(* IEC 61131-3 sources: brOscatLib/oscatNetw (part 6) *)

(* ---- SMTP_CLIENT.st ---- *)
FUNCTION_BLOCK SMTP_CLIENT
    (*http://www.oscat.de/images/OSCATNetwork/oscat_netlib121_en.pdf#page=123*)
    CASE step OF

    00:
    	IF ACTIVATE AND NOT activate_last THEN
    		TIMEOUT := MAX(T#10s,TIMEOUT);
    		timeout2 := TIMEOUT + T#1s;
    		timeout3 := TIMEOUT / 2;
    		DONE := FALSE;
    		ip_c_red_disable := FALSE;
    		ERROR_C := DWORD#0;
    		ERROR_T := BYTE#0;
    		FSD.ERROR := BYTE#0;
    		file_delete := FALSE;
    		URL_DATA := STRING_TO_URL(STR:=SERVER,DEFAULT_PROTOCOL:='',DEFAULT_PATH:='/');
    		idx1 := FIND(URL_DATA.USER,'%'); (* % Zeichen auf @ ändern *)
    		IF idx1 > 0 THEN
    			URL_DATA.USER := REPLACE(URL_DATA.USER,'@',1,idx1);
    		END_IF
    		esmtp := LEN(URL_DATA.PASSWORD) > 0; (* SMTP oder ExtendedSMTP *)
    		step := 10;
    	END_IF

    10:
    	IF DNS_CLIENT.DONE THEN
    		step := 20;
    	ELSIF DNS_CLIENT.ERROR <> DWORD#0 THEN
    		ERROR_C := DNS_CLIENT.ERROR;
    		ERROR_T := BYTE#1;
    		step := 980;
    	END_IF

    20:	(* SMTP Kommunikation einrichten *)
    	IF FIND(';SSL;ssl;Ssl', URL_DATA.PROTOCOL) > 1 THEN
    		ssl_mode := BYTE#1;
    		IP_C.C_PORT := SEL(URL_DATA.PORT = WORD#0,URL_DATA.PORT,WORD#465); (* Portnummer eintragen *)
    		IP_C.MAILBOX[16] := BYTE#1; (* SSL Mode freigeben *)
    	ELSIF FIND(';TLS;tls;Tls', URL_DATA.PROTOCOL) > 1 THEN
    		ssl_mode := BYTE#2;
    		IP_C.C_PORT := SEL(URL_DATA.PORT = WORD#0,URL_DATA.PORT,WORD#587); (* Portnummer eintragen *)
    		IP_C.MAILBOX[16] := BYTE#0; (* noch kein SSL Mode*)
    	ELSE
    		ssl_mode := BYTE#0;
    		IP_C.C_PORT := SEL(URL_DATA.PORT = WORD#0,URL_DATA.PORT,WORD#25); (* Portnummer eintragen *)
    		IP_C.MAILBOX[16] := BYTE#0; (* kein SSL Mode*)
    	END_IF

      	IP_C.C_IP := DNS_CLIENT.IP4; (* IP eintragen *)
      	IP_C.C_MODE := BYTE#0; (* Mode: TCP+ACTIV+PORT *)
      	IP_C.TIME_RESET := TRUE; (* Zeitueberwachung rücksetzen *)
      	IP_C.C_ENABLE := TRUE; (* Verbindungsaufbau freigeben *)
      	IP_C.R_OBSERVE := TRUE; (* Empfangsueberwachung *)
    	IP_C.MAILBOX[3] := BYTE#0; (* IP Empfang wieder freigeben *)
    	R_BUF.SIZE := UINT#0;
    	snd_enable := TRUE; (* sofortiges senden erlauben *)
    	snd_idx := 0;
    	step := 30;

    30:
    	IF rcv_state = 220 THEN (* 220 = Service ready *)
    		IF esmtp THEN
    			snd_text := 'EHLO OSCAT'; (* ExtendedSMTP *)

    			str1:= SEL(ssl_mode = BYTE#2,auth_names,auth_names_tls);
    			auth_state := BYTE#0;
    			idx2 := 1900;

    			next_step := 40;
    		ELSE
    			snd_text := 'HELO OSCAT'; (* SMTP *)
    			next_step := 90;
    		END_IF
    		snd_lf_cnt := 1;
    	END_IF

    40:
    	IF rcv_state = 250 THEN
    		(* 250 = Requested mail action okay, complete
    			1. bei manchen Providern wird bei SSL kein AUTH verfahren ausgeben.
    			2. Da die 250 xxx Meldungen vom manchen SMTP-Servern mit mehr als einem Telegramme versendet
    		       werden muss alternativ über Zeitüberwachung eine SSL Sonderbehandlung durchgeführt werden *)
    		IF ssl_mode >= BYTE#1 AND TON_WAIT.ET > T#1s THEN
    			rcv_text := '250-AUTH LOGIN'; (* AUTH vortäuschen *)

            	(*####################  DEBUG-MESSAGE  ###################################*)
    			(*IF _debug_enable THEN
    				LOG_CL.NEW_MSG := 'SMTP: PROBLEM /rcv_text ~1';
    				LOG_CL.PRINTF[1] := rcv_text;
    				LOG_MSG();
    			END_IF*)
    			(*########################################################################*)

    		END_IF

    		IF FIND(rcv_text,'AUTH') > 0 THEN (* BUGFIX  !*)
    			IP_C.MAILBOX[3] := BYTE#1; (* IP Empfang blockieren bis Daten überprüft wurden *)
    			idx1 := 0;
    			step := 50;
    		END_IF

    	END_IF

    50:
    	str2 := ELEMENT_GET(59, idx1, str1); (* Trennzeichen >;< *)

    	(*####################  DEBUG-MESSAGE  ###################################*)
    	(*IF _debug_enable THEN
    		LOG_CL.NEW_MSG := 'ST s1>~1< s2>~2< i1>~2< ~3';
    		LOG_CL.PRINTF[1] := str1;
    		LOG_CL.PRINTF[2] := str2;
    		LOG_CL.PRINTF[3] := INT_TO_STRING(idx1);
    		LOG_CL.PRINTF[4] := rcv_text;
    		LOG_MSG();
    	END_IF*)
    	(*########################################################################*)

    	IF LEN(str2) > 0 THEN
    		IF FIND(rcv_text,str2) > 0 THEN
    			auth_state := BIT_LOAD_B(auth_state, TRUE, idx1);
    			str3 := str2; (* aktuellen AUTH-Type Namen sichern *)
    			idx2 := 1000 + (idx1 * 100); (* Schritt berechnen *)
    		END_IF
    		idx1 := idx1 + 1;
    	ELSE
    		IF auth_state <> BYTE#0 THEN (* AUTH-Type gefunden *)
    			IP_C.MAILBOX[3] := BYTE#0; (* IP Empfang wieder freigeben *)
    			(* mit den jeweiligen Authentifizierung Schritten fortfahren:
    			   1000 = PLAIN / 1100 = LOGIN / 1200 = CRAM-MD5 / 1300 TLS *)
    			step := idx2;
    		ELSE
    			idx1 := 0;
    			rcv_text := '';
    			IP_C.MAILBOX[3] := BYTE#0; (* IP Empfang wieder freigeben *)
    			step := 40; (* warten auf nächste 250 auth meldung *)
    		END_IF
    	END_IF

    	(*####################  DEBUG-MESSAGE  ###################################*)
    	(*IF _debug_enable THEN
    		LOG_CL.NEW_MSG := 'SMTP: /auth ~1 /idx1 ~2 /idx2 ~3 /str3 ~4 /LEN ~5 /step ~6 /str1 ~7';
    		LOG_CL.PRINTF[1] := BYTE_TO_STRING(auth_state);
    		LOG_CL.PRINTF[2] := INT_TO_STRING(idx1);
    		LOG_CL.PRINTF[3] := INT_TO_STRING(idx2);
    		LOG_CL.PRINTF[4] := str3;
    		LOG_CL.PRINTF[5] := INT_TO_STRING(LEN(str2));
    		LOG_CL.PRINTF[6] := INT_TO_STRING(step);
    		LOG_CL.PRINTF[7] := str1;
    		LOG_MSG();
    	END_IF*)
    	(*########################################################################*)

     (* ++++++++++++++++++++++++++++++++++++++++++++++++++++++*)

    90:
    	IF rcv_state = 235 OR rcv_state = 250 THEN (* 235 = Authentication successful / 250 Requested mail action okay *)
    		str2 := MAILFROM;
    		str1 := ELEMENT_GET(59, 0, str2);(* MAILFROM lesen , Trennzeichen >;< *)
    		snd_text := INSERT('MAIL FROM: <>', str1, 12);
    		str3 := REPLACE(snd_text, 'From', 9, 1); (* 'MAIL FROM' durch "From" ersetzen und zwischenspeichern *)
    		next_step := 95;
    		cnt1 := ELEMENT_COUNT(35, MAILTO); (* Trennzeichen >#< , Anzahl der Blöcke bestimmen *)
    		cnt2 := 0;
    	END_IF

    95:
    	IF rcv_state = 250 THEN (* 250 = Requested mail action okay *)
    		IF cnt2 < cnt1 THEN
    			str1 := ELEMENT_GET(35, cnt2, MAILTO);(* Trennzeichen >#< *)
    			cnt3 := ELEMENT_COUNT(59, str1); (* Trennzeichen >;< , Anzahl der Sub-Blöcke bestimmen *)
    			cnt4 := 0;
    			cnt2 := cnt2 + 1;
    			step := 100; (* Blockinhalt auswerten *)
    		ELSE
    			step := 110; (* alle Blöcke bearbeitet *)
    		END_IF
    	END_IF

    100:
    	IF rcv_state = 250 THEN (* 250 = Requested mail action okay *)
    		IF cnt4 < cnt3 THEN
    			str2 := ELEMENT_GET(59, cnt4, str1); (* Trennzeichen >;< *)
    			snd_text := INSERT('RCPT TO: <>', str2, 10);
    			cnt4 := cnt4 + 1;
    			next_step := 100;
    		ELSE
    			step := 95;
    		END_IF
    	END_IF

    110:
    	IF rcv_state = 250 THEN (* 250 = Requested mail action okay *)
    		snd_text := 'DATA';
    		next_step := 120;
    	END_IF

    120:
    	IF rcv_state = 354 THEN (* 354 = Start mail input; end with. *)
    		snd_enable := FALSE;
    		str2 := MAILFROM;
    		str1 := ELEMENT_GET(59, 1, str2);(* Angezeigter Name lesen , Trennzeichen >;< *)
    		IF LEN(str1) > 0 THEN
    			str2 := INSERT('"" ', str1, 1);
    			snd_text := INSERT(str3, str2, 6);
    		ELSE
    			snd_text := str3;
    		END_IF
    		cnt2 := 0;
    		cnt1 := MIN(2,cnt1); (* BlindCopy Block ausblenden *)
    		step := 200;
    	END_IF

    200:
    	IF snd_step = 0 THEN
    		IF cnt2 < cnt1 THEN
    			str1 := ELEMENT_GET(35, cnt2, MAILTO);(* Trennzeichen >#< *)
    			cnt3 := ELEMENT_COUNT(59, str1); (* Trennzeichen >;< , Anzahl der Sub-Blöcke bestimmen *)
    			cnt4 := 0;
    			cnt2 := cnt2 + 1;
    			str3 := SEL(cnt2 = 1,'Cc: <>','To: <>');
    			step := 205; (* Blockinhalt auswerten *)
    		ELSE
    			step := 210; (* alle Blöcke bearbeitet *)
    		END_IF
    	END_IF

    205:
    	IF snd_step = 0 THEN
    		IF cnt4 < cnt3 THEN
    			str2 := ELEMENT_GET(59, cnt4, str1); (* Trennzeichen >;< *)
    			snd_text := INSERT(str3, str2, 5);
    			cnt4 := cnt4 + 1;
    		ELSE
    			step := 200;
    		END_IF
    	END_IF

    210:
    	IF snd_step = 0 THEN
    		snd_text := CONCAT('SUBJECT: ',SUBJECT);
    		step := 220;
    	END_IF

    220:
    	IF snd_step = 0 THEN
    		DTI := UDINT_TO_DT(DT_TO_UDINT(DTI) + INT_TO_UDINT(- DTI_OFFSET * 60)); (* Minuten-Offset auf Sekunden umrechnen und addieren *)
    		IF esmtp THEN (* esmtp Format >Date: Thu, 21 May 1998 05:33:29 -0700< *)
    			str2 := ';Mon;Tue;Wed;Thu;Fri;Sat;Sun';
    			str1 := ELEMENT_GET(59, DAY_OF_WEEK(DT_TO_DATE(DTI)), str2);
    			snd_text := CONCAT('Date: ',str1);
    			str1 := DT_TO_STRF(DTI, 0, ', #H #E #A #N:#R:#T +0000', 1);
    			snd_text := CONCAT(snd_text,str1);
    		ELSE (* SMTP Format >Date: 21 May 98 05:33:29< *)
    			snd_text := DT_TO_STRF(DTI, 0, 'Date: #G #E #B #N:#R:#T', 1);
    		END_IF
    		step := 230;
    	END_IF

    230:
    	IF snd_step = 0 THEN
    		snd_text := 'MIME-Version: 1.0';
    		step := 250;
    	END_IF

    250:
    	IF snd_step = 0 THEN
    		snd_text := 'Content-Type: multipart/mixed;boundary="x"';
    		snd_lf_cnt := 2;
    		step := 260;
    	END_IF

    260:
    	IF snd_step = 0 THEN
    		snd_enable := TRUE;
    		snd_text := 'This is a multi-part message in MIME format.';
    		step := 270;
    	END_IF

    270:
    	IF snd_step = 0 THEN
    		snd_enable := FALSE;
    		snd_text := '--x';
    		snd_lf_cnt := 1;
    		step := 280;
    	END_IF

    280:
    	IF snd_step = 0 THEN
    		snd_text := 'Content-Type: text/plain; format=flowed; charset="iso-8859-1";';
    		snd_text := CONCAT(snd_text,' reply-type=original'); (* PCWORX kann nur konstanten mit max 80 zeichen *)
    		step := 290;
    	END_IF

    290:
    	IF snd_step = 0 THEN
    		snd_text := 'Content-Transfer-Encoding: 8bit';
    		snd_lf_cnt := 2;
    		step := 300;
    	END_IF

    300:
    	IF snd_step = 0 THEN
    		snd_enable := TRUE;
    		snd_text := BODY;
    		snd_lf_cnt := 2;
    		step := 310;
    	END_IF

    310:
    	IF snd_step = 0 THEN
    		cnt1 := ELEMENT_COUNT(59, FILES) - 1; (* Anzahl der Dateien *)
    		step := 400;
    	END_IF

    (* +++++++++++++ File-Attachment ++++++++++++ *)
    400:
    	IF cnt1 >= 0 THEN
    		str1 := ELEMENT_GET(59, cnt1, FILES);
    		FILE_PATH_SPLIT(FILENAME:=str1,X:=fpd); (* Datei-Path zerlegen *)
    		IF fpd.FILENAME = '#DEL#' THEN
    			file_delete := TRUE;
    		ELSE
    			step := 410;
    		END_IF
    		cnt1 := cnt1 - 1;
    	ELSE
    		step := 800;
    	END_IF

    410:
    	IF snd_step = 0 THEN
    		snd_enable := FALSE;
    		snd_text := '--x';
    		snd_lf_cnt := 1;
    		step := 420;
    	END_IF

    420:
    	IF snd_step = 0 THEN
    		snd_text := 'Content-Transfer-Encoding: BASE64';
    		str2 := CONCAT(fpd.FILENAME,'"');
    		step := 430;
    	END_IF

    430:
    	IF snd_step = 0 THEN
    		snd_text := CONCAT('Content-Type: application/octet-stream; name="',str2);
    		step := 440;
    	END_IF

    440:
    	IF snd_step = 0 THEN
    		snd_enable := TRUE;
    		snd_text := CONCAT('Content-Disposition: attachment; filename="',str2);
    		snd_lf_cnt := 2;
    		step := 450;
    	END_IF

    450:
    	IF snd_step = 0 THEN
    		FSD.FILENAME := str1; (* Dateiname *)
    		FSD.OFFSET := UDINT#0; (* Start bei Dateianfang *)
    		step := 460;
    	END_IF

    460:
    	FSD.MODE := BYTE#1; (* vorhandene Datei zum lesen öffnen *)
    	F_BUF.SIZE := b64_max; (* maximale länge einlesen *)
    	idx1 := 0;
    	idx2 := 0;
    	step := 470;

    470:
    	IF FSD.MODE = BYTE#0 AND FSD.ERROR = BYTE#0 THEN
    		last_block := FSD.FILE_SIZE = FSD.OFFSET;
    		b64_size1 := MIN(48,UINT_TO_INT(F_BUF.SIZE) - idx1);
    		IF b64_size1 > 0 THEN
    			idx3 := b64_size1 - 1;
    			FOR i1 := 0 TO idx3 DO (* daten in BASE64 buffer kopieren *)
    				b64_buf1[i1] := F_BUF.BUFFER[idx1];
    				idx1 := idx1 + 1;
    			END_FOR
    			BASE64_ENCODE_STREAM( SIZE1:= b64_size1, BUF1:= b64_buf1, BUF2:= b64_buf2, SIZE2=> b64_size2); (* BASE64 Kodierung *)
    			idx3 := b64_size2 - 1;
    			FOR i1 := 0 TO idx3 DO (* Daten aus BASE64 buffer kopieren *)
    				S_BUF.BUFFER[idx2] := b64_buf2[i1];
    				idx2 := idx2 + 1;
    			END_FOR
    			b64_lf := TRUE;
    			(*####################  DEBUG-MESSAGE  ###################################*)
    			(*IF _debug_enable THEN
    				LOG_CL.NEW_MSG := 'B64: FILE ~1 /SIZE ~2 /OFF ~3 /BSIZE ~4 /idx1 ~5 /idx2 ~6';
    				LOG_CL.PRINTF[1] := FSD.FILENAME;
    				LOG_CL.PRINTF[2] := UDINT_TO_STRING(FSD.FILE_SIZE);
    				LOG_CL.PRINTF[3] := UDINT_TO_STRING(FSD.OFFSET);
    				LOG_CL.PRINTF[4] := INT_TO_STRING(b64_size1);
    				LOG_CL.PRINTF[5] := INT_TO_STRING(idx1);
    				LOG_CL.PRINTF[6] := INT_TO_STRING(idx2);
    				LOG_MSG();
    			END_IF*)
    			(*########################################################################*)
    		ELSE
    			b64_lf := last_block;
    			step := 480; (* block beendet  *)
    		END_IF
    		IF b64_lf THEN
    			S_BUF.BUFFER[idx2] := BYTE#16#0D;
    			idx2 := idx2 + 1;
    			S_BUF.BUFFER[idx2] := BYTE#16#0A;
    			idx2 := idx2 + 1;
    		END_IF
    		(*####################  DEBUG-MESSAGE  ###################################*)
    		(*IF _debug_enable THEN
    			LOG_CL.NEW_MSG := 'B64: exit ~1 /SIZE ~2 /OFF ~3 /eof ~4 /lf_cnt ~5';
    			LOG_CL.PRINTF[1] := FSD.FILENAME;
    			LOG_CL.PRINTF[2] := UDINT_TO_STRING(FSD.FILE_SIZE);
    			LOG_CL.PRINTF[3] := UDINT_TO_STRING(FSD.OFFSET);
    			LOG_CL.PRINTF[4] := BOOL_TO_STRING(last_block);
    			LOG_CL.PRINTF[5] := INT_TO_STRING(snd_lf_cnt);
    			LOG_MSG();
    		END_IF*)
    		(*########################################################################*)
    	END_IF

    480:
    	S_BUF.SIZE := INT_TO_UINT(idx2); (* Daten senden *)
    	(*####################  DEBUG-MESSAGE  ###################################*)
    	(*IF _debug_enable THEN
    		LOG_CL.NEW_MSG := 'B64: tcp_send ~1';
    		LOG_CL.PRINTF[1] := INT_TO_STRING(idx2);
    		LOG_MSG();
    	END_IF*)
    	(*########################################################################*)
    	step := 490;

    490:
    	IF S_BUF.SIZE = UINT#0 THEN (* warten bis alle daten gesendet sind *)
    		step := SEL(last_block ,460,400);
    	END_IF

    (* ++++++++++++++++++++++++++++++++++++++++ *)

    800:
    	IF snd_step = 0 THEN
    		snd_enable := FALSE;
    		snd_text := '--x--';
    		snd_lf_cnt := 2;
    		step := 810;
    	END_IF

    810:
    	IF snd_step = 0 THEN
    		snd_enable := TRUE;
    		snd_text := '.';
    		snd_lf_cnt := 1;
    		step := 820;
    	END_IF

    820:
    	IF rcv_state = 250 THEN (* 250 = Requested mail action okay *)
    		snd_text := 'QUIT';
    		ip_c_red_disable := TRUE;
    		next_step := 830;
    	END_IF

    830:
    	IF rcv_state = 221  OR TON_WAIT.ET > timeout3 THEN (* 221 = Service closing transmission channel *)
    		step := 900;
    	END_IF

    (* ================================================== *)

    900:
    	IF file_delete THEN (* Dateien nach transfer löschen *)
    		cnt1 := ELEMENT_COUNT(59, FILES) - 1; (* Trennzeichen >;< , Anzahl der Dateien *)
    		step := 910;
    	ELSE
    		step := 950;
    	END_IF

    910:
    	IF FSD.MODE = BYTE#0 AND FSD.ERROR = BYTE#0 THEN
    		IF cnt1 >= 0 THEN
    			str1 := ELEMENT_GET(59, cnt1, FILES); (* Trennzeichen >;< *)
    			IF str1 <> '#DEL#' THEN
    				FSD.FILENAME := str1;
    				FSD.MODE := BYTE#4; (* File Remove *)
    			END_IF
    			cnt1 := cnt1 - 1;
    		ELSE
    			step := 950;
    		END_IF
    	END_IF

    950:
    	DONE := TRUE;
    	step := 980;

    980:
    	IP_C.C_ENABLE := FALSE; (* SMTP Steuerkanal schliessen *)
    	S_BUF.SIZE := UINT#0;
    	R_BUF.SIZE := UINT#0;
    	IP_C.MAILBOX[3] := BYTE#0; (* IP Empfang wieder freigeben *)
    	snd_step := 0;
    	next_step := 0;
    	FSD.MODE := BYTE#5; (* Datei schliessen *)
    	step := 990;

    990:
    	IF IP_C.C_STATE = BYTE#0 AND FSD.FILE_OPEN = FALSE THEN
    		step := 0;
    	END_IF

    (*  +++++++++++++++++ Authentifizierung +++++++++++++++++ *)

    (* PLAIN ++++++++++++++++++++++++++++++++++++++++++++++++++++++++++ *)

    1000:
    	snd_text := CONCAT('AUTH',str3);
    	snd_lf_cnt := 1;
     	step := 1010;

    1010:
    	IF rcv_state = 334 THEN (* 334 = Authentifizierung  *)
    		cnt1 := LEN(URL_DATA.USER);
    		cnt2 := LEN(URL_DATA.PASSWORD);
    		IF cnt1 + cnt2 <= 46 THEN (* USER + PASSWORD dürfen zusammen maximal 46 Zeichen haben *)
    			b64_buf1[0] := BYTE#0;
    			FOR i1 := 1 TO cnt1 DO
    				b64_buf1[i1] := CODE(URL_DATA.USER, i1);
    			END_FOR
    			b64_size1 := cnt1 + 1;
    			b64_buf1[b64_size1] := BYTE#0;
    			b64_size1 := b64_size1 + 1;
    			FOR i1 := 1 TO cnt2 DO
    				b64_buf1[b64_size1] := CODE(URL_DATA.PASSWORD, i1);
    				b64_size1 := b64_size1 + 1;
    			END_FOR
    			BASE64_ENCODE_STREAM( SIZE1:= b64_size1, BUF1:= b64_buf1, BUF2:= b64_buf2, SIZE2=> b64_size2); (* BASE64 Kodierung *)
    			idx1 := b64_size2 - 1;
    			FOR i1 := 0 TO idx1 DO
    				S_BUF.BUFFER[i1] := b64_buf2[i1];
    			END_FOR
    			S_BUF.BUFFER[b64_size2] := BYTE#16#0D;
    			b64_size2 := b64_size2 + 1;
    			S_BUF.BUFFER[b64_size2] := BYTE#16#0A;
    			b64_size2 := b64_size2 + 1;
    			S_BUF.SIZE := INT_TO_UINT(b64_size2);
    			rcv_state := 0;
    		END_IF
    		step := 90;
    	END_IF

    (* LOGIN ++++++++++++++++++++++++++++++++++++++++++++++++++++++++++ *)

    1100:
    	snd_text := CONCAT('AUTH',str3);
    	snd_lf_cnt := 1;
     	step := 1110;

    1110:
    	IF rcv_state = 334 THEN (* 334 = Authentifizierung  *)
    		b64_str1 := URL_DATA.USER;
    		b64_start := TRUE; (* BASE64 kodierung von Username *)
    		step := 1120;
    	END_IF

    1120:
    	IF b64_start AND b64_done THEN
    		b64_start := FALSE;
    		snd_text := b64_str2;
    		next_step := 1130;
    	END_IF

    1130:
    	IF rcv_state = 334 THEN (* 334 = Password:  *)
    		b64_str1 := URL_DATA.PASSWORD;
    		b64_start := TRUE; (* BASE64 kodierung von Password *)
    		step := 1140;
    	END_IF

    1140:
    	IF b64_start AND b64_done THEN
    		b64_start := FALSE;
    		snd_text := b64_str2;
    		next_step := 90;
    	END_IF

    (* CRAM-MD5  ++++++++++++++++++++++++++++++++++++++++++++++++++++++++++
    (Challenge-Response Authentication Mechanism, Message Digest 5) Authentifizierung auf Basis von MD5-HMAC-Algorithmus. *)

    1200:
    	snd_text := CONCAT('AUTH',str3);
    	snd_lf_cnt := 1;
     	step := 1210;

    1210:
    	IF rcv_state = 334 THEN (* 334 = Authentifizierung  *)
    		md5_b64_ts := RIGHT(rcv_text,LEN(rcv_text) - 4);
    		md5_user := URL_DATA.USER;
    		md5_password := URL_DATA.PASSWORD;
    		MD5_RUN := TRUE;
    		step := 1220;
    	END_IF

    1220:
    	MD5_CRAM_AUTH(RUN:=MD5_RUN,USERNAME:=md5_user,PASSWORD:=md5_password,B64_TS:=md5_b64_ts,AUTH_KEY:=md5_auth_key);
    	IF NOT MD5_RUN THEN
    		snd_text := md5_auth_key;
    		step := 90;
    	END_IF

    (* STARTTLS  ++++++++++++++++++++++++++++++++++++++++++++++++++++++++++ *)

    1300:
    	snd_text := 'STARTTLS';
    	snd_lf_cnt := 1;
     	step := 1310;

    1310:
    	IF rcv_state = 220 THEN (* 220 = Service ready - Ready to start TLS *)
    		IP_C.MAILBOX[16] := BYTE#1; (* SSL/TLS aktivieren *)
    		step := 1320;
    	END_IF

    1320:
    	IF IP_C.MAILBOX[16] = BYTE#2 THEN (* warten bis SSL/TLS aktiviert wurde *)
    		step := 30; (* ganzer Ablauf von vorne beginnen *)
    	END_IF

    (* keine Authentifizierung gefunden +++++++++++++++++++++++++++++++ *)
    1900: ; (* Auf Laufzeitfehler warten *)

    END_CASE
    (* ++++++++++++++++++++++++++++++++++++++++++++++++++++++++++ *)
    IF step >= 30 THEN
    	IF R_BUF.SIZE > UINT#0 THEN (* Daten wurden empfangen ? *)
    		idx1 := UINT_TO_INT(R_BUF.SIZE);
    		REPEAT (* zeilenterminierung erkennen und echtes TEXT-Ende bestimmen *)
    			idx1 := idx1 - 1;
    		UNTIL idx1 = 0 OR R_BUF.BUFFER[idx1] >= BYTE#32 (* TRUE = EXIT *)
    		END_REPEAT
    		FOR i1 := 0 TO idx1 DO (* bei multiline alle CRLF durch >< ersetzen *)
    			IF R_BUF.BUFFER[i1] < BYTE#32 THEN
    				R_BUF.BUFFER[i1] := BYTE#94; (* >< *)
    			END_IF
    		END_FOR
    		rcv_text := BUFFER_TO_STRING(PT:=ADR(R_BUF.BUFFER),SIZE:=idx1+1,START:=0,STOP:=STRING_LENGTH-1);
    		IF LEN(rcv_text) >= 3 THEN (* Statuscode prüfen und auswerten *)
    			rcv_s := LEFT(rcv_text,3);
    			IF IS_NUM(STR:=rcv_s) THEN (* enthält nur Zahlen ? *)
    				rcv_state := STRING_TO_INT(rcv_s);
    			END_IF
    			IP_C.R_OBSERVE := FALSE;
    		END_IF
    		R_BUF.SIZE := UINT#0; (* daten löschen *)

    		(*####################  DEBUG-MESSAGE  ###################################*)
    		(*IF _debug_enable THEN
    			LOG_CL.NEW_MSG := 'RCV: >~1<';
    			LOG_CL.PRINTF[1] := rcv_text;
    			LOG_MSG();
    		END_IF*)
    		(*########################################################################*)

    	END_IF
    END_IF

    (* automatisches Datensenden *)

    CASE snd_step OF

    00:
    	IF LEN(snd_text) > 0 THEN

    		(*####################  DEBUG-MESSAGE  ###################################*)
    		(*IF _debug_enable THEN
    			LOG_CL.NEW_MSG := 'SND: >~1< /lf ~2';
    			LOG_CL.PRINTF[1] := snd_text;
    			LOG_CL.PRINTF[2] := INT_TO_STRING(snd_lf_cnt);
    			LOG_MSG();
    		END_IF*)
    		(*########################################################################*)

    		_STRING_TO_BUFFER(str:=snd_text,pos:=snd_idx,pt:=ADR(S_BUF.BUFFER),size:=SIZEOF(S_BUF.BUFFER)); (* String in puffer kopieren *)
    		snd_idx := snd_idx + LEN(snd_text);
    		FOR i1 := 1 TO snd_lf_cnt DO
    			S_BUF.BUFFER[snd_idx] := BYTE#16#0D;
    			snd_idx := snd_idx + 1;
    			S_BUF.BUFFER[snd_idx] := BYTE#16#0A;
    			snd_idx := snd_idx + 1;
    		END_FOR
    		snd_text := '';
    		rcv_state := 9999; (* letzen SMTP Status löschen *)

    		IF snd_enable THEN
    			S_BUF.SIZE := INT_TO_UINT(snd_idx); (* Sendelänge eintragen *)
    			R_BUF.SIZE := UINT#0; (* Empfangsbuffer rücksetzen *)
    			IP_C.R_OBSERVE := step <= 120 OR step >= 820;
    			snd_idx := 0;
    			snd_step := 10;
    		END_IF
    	END_IF

    10:
    	IF S_BUF.SIZE = UINT#0 THEN (* warten bis alle daten gesendet sind *)
    		IF next_step <> 0 THEN
    			step := next_step;
    			next_step := 0;
    		END_IF
    		snd_step := 0;
    	END_IF

    END_CASE

    (* Globale Fehlerbehandlung für Haupt-Routine *)
    IF ERROR_T = BYTE#0 AND step > 20 THEN (* noch kein Fehler gespeichert und Hauptroutine aktiv *)

    	IF IP_C.ERROR > DWORD#0 AND IP_C.C_ENABLE AND NOT IP_C.TIME_RESET THEN  (* IP Control 1 *)
    		IF ip_c_red_disable = FALSE OR IP_C.ERROR <> DWORD#16#FD000000 THEN
    			ERROR_C := IP_C.ERROR;
    			ERROR_T := BYTE#2;
    			step := 980;
    		END_IF
    	END_IF

    	IF FSD.MODE = BYTE#0 THEN
    		IF FSD.ERROR > BYTE#0 THEN
    			ERROR_C := BYTE_TO_DWORD(FSD.ERROR);
    			ERROR_T := BYTE#4; (* Dateizugriff *)
    			step := 980;
    		END_IF
    	END_IF
    END_IF

    IF TON_WAIT.Q THEN (* Ablaufstörung - Schrittkette *)
    	ERROR_C := SHL(INT_TO_DWORD(step),16) OR INT_TO_DWORD(rcv_state); (* aktuellen Schritt und letzten SMTP Status eintragen *)
    	ERROR_T := BYTE#5;
    	step := 980;
    END_IF

    (* ######################################################## *)

    DNS_CLIENT(IP_C:=IP_C, S_BUF:=S_BUF, R_BUF:=R_BUF, DOMAIN:=URL_DATA.DOMAIN, IP4_DNS:= DNS_IP4, ACTIVATE:=step=10); (* DNS-Client *)
    IPC(IP:= DWORD#0, PORT:= WORD#0 , TIME_OUT:= TIMEOUT, IP_C:= IP_C, S_BUF:= S_BUF, R_BUF:= R_BUF); (* SMTP Steuerkanal *)
    FS(FSD:=FSD,PT:=F_BUF); (* FILE_SERVER *)
    BASE64_ENCODE_STR(RUN:= b64_start, str1:= b64_str1, str2:= b64_str2, DONE=> b64_done); (* BASE64 kodierung *)

    TON_WAIT(IN:=step = last_step AND step > 0,PT:=timeout2);
    last_step := step;
    activate_last := ACTIVATE;
    BUSY := step <> 0;

    (* revision history
    ks	01. jan. 2011	rev 1.0
    	original version
    ks	06. apr. 2011	rev 1.1
    	list_len und list_get durch element_count und element_get ersetzt
    ks	11. may 2011	rev 1.2
    	ip_control - remote disconnect error ausblenden, und sonderbehandlung für pcworx
    ks	30. may 2011	rev 1.3
    	fehler bei receive-TIMEOUT
    ks	05. may. 2012	rev 1.4
    	FileServer AutoClose entfernt und Fehler im Alias Name korrigiert
    ks	06. apr. 2013	rev 1.5
    	Fehler bei Authorisierungsabfrage bei 1&1 Provider behoben
    ks	22. feb. 2016	rev 1.6
    	integration SSL/TLS
    ks	11. aug. 2016	rev 1.7
    	bugfix: Find SSL/TLS String in URL_DATA.PROTOCOL
    *)
END_FUNCTION_BLOCK

(* ---- SNTP_CLIENT.st ---- *)
FUNCTION_BLOCK SNTP_CLIENT
    (*http://www.oscat.de/images/OSCATNetwork/oscat_netlib121_en.pdf#page=127*)
    (* Domain Name System (query) *)
    tx := T_PLC_MS(); (* read system time *)

    CASE state OF
    00: (* auf positive Flanke SET warten *)
    	DONE_P := FALSE;
    	IF ACTIVATE AND NOT activate_last THEN
    		ip4_stored := IP4; (* aktuelle IP4 speichern *)
    		state := 10;
    		ERROR := DWORD#0;
    		ip_state := BYTE#1; (* Anmelden *)
    		(*####################  DEBUG-MESSAGE  ###################################*)
    		(*IF _debug_enable THEN
    			LOG_CL.NEW_MSG := 'SNTP: S00 START';
    			LOG_MSG();
    		END_IF*)
    		(*########################################################################*)
    	END_IF

    10: (* Bei IP_Control anmelden und auf freigabe warten *)
    	IF ip_state = BYTE#3 THEN

    		S_BUF.BUFFER[00] := BYTE#16#1B;
    		FOR i := 1 TO 47 DO
    			S_BUF.BUFFER[i] := BYTE#16#00;
    		END_FOR

    		last := tx; (* aktuellen time wert sichern *)
    		state := 30;

    		(* IP Datenverkehr einrichten *)
    		IP_C.C_PORT := WORD#123; (* Portnummer eintragen *)
    		IP_C.C_IP := ip4_stored; (* IP eintragen *)
    		IP_C.C_MODE := BYTE#1; (* Mode: UDP+AKTIV+PORT+IP *)
    		IP_C.C_ENABLE := TRUE; (* Verbindungsaufbau freigeben *)
    		IP_C.TIME_RESET := TRUE; (* Zeitueberwachung rücksetzen *)
    		IP_C.R_OBSERVE := TRUE; (* Datenempfang ueberwachen *)
    		S_BUF.SIZE := UINT#48; (* Sendelänge eintragen *)
    		R_BUF.SIZE := UINT#0; (* Empfangslänge rücksetzen *)
        		(*####################  DEBUG-MESSAGE  ###################################*)
        		(*IF _debug_enable THEN
          			LOG_CL.NEW_MSG := 'SNTP: S10 SEND';
          			LOG_MSG();
        		END_IF*)
        		(*########################################################################*)
    	END_IF

    30:
    	IF IP_C.ERROR <> DWORD#00 THEN
    		ERROR := IP_C.ERROR;
    		S_BUF.SIZE := UINT#0;
    		R_BUF.SIZE := UINT#0;
    		state := 0;
        		(*####################  DEBUG-MESSAGE  ###################################*)
        		(*IF _debug_enable THEN
          			LOG_CL.NEW_MSG := 'SNTP: S30 ERROR ~1';
          			LOG_CL.PRINTF[1] := DWORD_TO_STRING(ERROR);
          			LOG_MSG();
        		END_IF*)
        		(*########################################################################*)

    	ELSIF S_BUF.SIZE = UINT#0 AND R_BUF.SIZE >= UINT#48 THEN (* länge der empfangenen Daten prüfen *)

    		(* Umrechnung SNTP Timestamp Base 1900-01-01 -> Unix 1970-01-01 = +2208988800 sekunden*)
    		UDT := DWORD_TO_DT(DWORD_OF_BYTE(R_BUF.BUFFER[40],R_BUF.BUFFER[41],R_BUF.BUFFER[42],R_BUF.BUFFER[43]) - DWORD#2208988800);

    		(* Original-Sekundenanteile sind als 32 Bit Fractal dargestellt *)
    		(* ms nur mit veringerte Auflösung berechnen 1/65535 -> Highword verwenden *)
    		XMS := DWORD_TO_INT(SHR(DINT_TO_DWORD(WORD_TO_DINT(WORD_OF_BYTE(R_BUF.BUFFER[44],R_BUF.BUFFER[45])) * DINT#1000),16));
    		(* Zeitdifferenz (Laufzeitfehler) zwischen Send und Receive /2 teilen und addieren *)
    		XMS := XMS + DWORD_TO_INT(SHR(tx - last,1));

    		UDT := DWORD_TO_DT(DT_TO_DWORD(UDT) + (XMS / 1000)); (* sekundenanteile der Zeitdifferenz zu UDT aufrechnen *)
    		XMS := XMS MOD 1000;  (* ms übernehmen *)
    		state := 0;
    		DONE_P := TRUE;
        		(*####################  DEBUG-MESSAGE  ###################################*)
        		(*IF _debug_enable THEN
            			LOG_CL.NEW_MSG := 'SNTP: S30 OK';
            			LOG_MSG();
        		END_IF*)
        		(*########################################################################*)

    	END_IF

    	IF state = 0 THEN
    		IP_C.R_OBSERVE := FALSE; (* Datenempfang ueberwachen *)
    		ip_state := BYTE#4;
    	END_IF

    END_CASE

    activate_last := ACTIVATE; (* letzten Status sichern zur Flankenerkennung *)

    (* IP_FIFO *)
    IP_FIFO(FIFO:=IP_C.FIFO,state:=ip_state,ID:=ip_id);

    (* revision history
    ks	18. oct. 2008	rev 1.0
    	original version

    ks	20. oct. 2009	rev 1.1
    	Networkbuffer und Buffer-funktionen auf Basis 0

    *)

    (***************************************************************************************)
    (*               SNTP Datenstruktur
                                      1                   2                   3
                  0 1 2 3 4 5 6 7 8 9 0 1 2 3 4 5 6 7 8 9 0 1 2 3 4 5 6 7 8 9 0 1
                 +-+-+-+-+-+-+-+-+-+-+-+-+-+-+-+-+-+-+-+-+-+-+-+-+-+-+-+-+-+-+-+-+
    Byte: 01-04  |LI | VN  |Mode |    Stratum    |     Poll      |   Precision   |
                 +-+-+-+-+-+-+-+-+-+-+-+-+-+-+-+-+-+-+-+-+-+-+-+-+-+-+-+-+-+-+-+-+
    Byte: 05-08  |                          Root  Delay (32 Bit)                 |
                 +-+-+-+-+-+-+-+-+-+-+-+-+-+-+-+-+-+-+-+-+-+-+-+-+-+-+-+-+-+-+-+-+
    Byte: 09-12  |                       Root  Dispersion (32 Bit)               |
                 +-+-+-+-+-+-+-+-+-+-+-+-+-+-+-+-+-+-+-+-+-+-+-+-+-+-+-+-+-+-+-+-+
    Byte: 13-16  |                     Reference Identifier (32 Bit)             |
                 +-+-+-+-+-+-+-+-+-+-+-+-+-+-+-+-+-+-+-+-+-+-+-+-+-+-+-+-+-+-+-+-+
    Byte: 17-24  |                    Reference Timestamp (64 Bit)               |
                 +-+-+-+-+-+-+-+-+-+-+-+-+-+-+-+-+-+-+-+-+-+-+-+-+-+-+-+-+-+-+-+-+
    Byte: 25-32  |                    Originate Timestamp (64 Bit)               |
                 +-+-+-+-+-+-+-+-+-+-+-+-+-+-+-+-+-+-+-+-+-+-+-+-+-+-+-+-+-+-+-+-+
    Byte: 33-40  |                     Receive Timestamp (64 Bit)                |
                 +-+-+-+-+-+-+-+-+-+-+-+-+-+-+-+-+-+-+-+-+-+-+-+-+-+-+-+-+-+-+-+-+
    Byte: 41-48  |                     Transmit Timestamp (64 Bit)               |
                 +-+-+-+-+-+-+-+-+-+-+-+-+-+-+-+-+-+-+-+-+-+-+-+-+-+-+-+-+-+-+-+-+
    Byte: 49-52  |                 Key Identifier (optional) (32 Bit)            |
                 +-+-+-+-+-+-+-+-+-+-+-+-+-+-+-+-+-+-+-+-+-+-+-+-+-+-+-+-+-+-+-+-+
    Byte: 53-68  |                 Message Digest (optional) (128 Bit)           |
                 +-+-+-+-+-+-+-+-+-+-+-+-+-+-+-+-+-+-+-+-+-+-+-+-+-+-+-+-+-+-+-+-+

    *)

    (*
    Worldwide NTP-Server

    NIST-Zeitserver
    • time-a.nist.gov
    129.6.15.28
    NIST, Gaithersburg, Maryland
    • time-a.nist.gov
    129.6.15.28
    NIST, Gaithersburg, Maryland
    • time-a.timefreq.bldrdoc.gov
    132.163.4.101 (Stand: 1. Dezember 1999)
    NIST, Boulder, Colorado
    • time-b.timefreq.bldrdoc.gov
    132.163.4.102 (Stand: 1. Dezember 1999)
    NIST, Boulder, Colorado
    • time-c.timefreq.bldrdoc.gov
    132.163.4.103 (Stand: 1. Dezember 1999)
    NIST, Boulder, Colorado
    • utcnist.colorado.edu
    128.138.140.44
    University of Colorado, Boulder
    • time.nist.gov
    192.43.244.18
    NCAR, Boulder, Colorado
    • time-nw.nist.gov
    131.107.1.10
    Microsoft, Redmond, Washington
    • nist1.dc.certifiedtime.com
    216.200.93.8
    Abovnet, North Virginia
    • nist1.datum.com
    209.0.72.7
    Datum, San Jose, Kalifornien
    • nist1.nyc.certifiedtime.com
    208.184.49.129
    Abovnet, New York City
    • nist1.sjc.certifiedtime.com
    207.126.103.202
    Abovnet, San Jose, Kalifornien

    Zeitserver der ersten Ebene
    Sortiert nach Standort:
    Nordamerika
    • Palo Alto, Kalifornien: Systems Research Center, Compaq Computer Corp.
    204.123.2.72: usno.pa-x.dec.com; CNAME: navobs1.pa-x.dec.com
    Servicebereich: US-Zeitzonen PST (Pacific Standard Time) und MST (Mountain Standard Time)
    • Marina del Rey, Kalifornien: USC Information Sciences Institute
    128.9.176.30: timekeeper.isi.edu
    Servicebereich: CalRen2- und Los Nettos-Bereich
    • Washington, DC: U.S. Naval Observatory
    192.5.41.41: tock.usno.navy.mil
    192.5.41.40: tick.usno.navy.mil
    Servicebereich: NSFNET
    • Ottawa, Ontario, Kanada: National Research Council of Canada
    time.chu.nrc.ca
    Servicebereich: Kanada
    • Raleigh, North Carolina: North Carolina state University
    152.1.58.124: terrapin.csc.ncsu.edu
    Servicebereich: Südosten der USA
    • Cambridge, Massachusetts: MIT Information Systems
    18.72.0.3: bitsy.mit.edu
    Servicebereich: NSFNET- und NEARnet-Bereich
    • Cambridge, Massachusetts: MIT
    18.26.4.105: bonehed.lcs.mit.edu
    Servicebereich: Osten der USA
    • Palo Alto, Kalifornien: Internet Software Consortium
    192.5.5.250: clock.isc.org
    Servicebereich: BARRnet, Alternet-West und CIX-West
    • Cambridge, Massachusetts: Open Software Foundation
    130.105.4.59: clock.osf.org
    Servicebereich: NSFNET- und NEARnet-Bereich
    • Palo Alto, Kalifornien: ViaNet Communications
    209.81.9.7: clock.via.net
    • Cleveland, Ohio: Lewis Research Center (NASA)
    128.156.1.43: lerc-dns.lerc.nasa.gov
    Servicebereich: NSFNET und OARNET
    • Colorado Springs, Colorado: Schriever AFB
    204.34.198.40: navobs1.usnogps.navy.mil; CNAME: tick.usnogps.navy.mil
    204.34.198.41: navobs1.usnogps.navy.mil; CNAME: tock.usnogps.navy.mil
    Servicebereich: US-Zeitzonen PST (Pacific Standard Time) und MST (Mountain Standard Time)
    • St. Louis, Missouri: Washington University
    128.252.19.1: navobs1.usnogps.navy.mil; CNAME: tick.wustl.edu
    Servicebereich: US-Zeitzone CST (Central Standard Time)
    • Research Triangle Park, North Carolina: MCNC
    192.101.21.1: ncnoc.ncren.net
    Servicebereich: NC-REN-Bereich (North Carolina Research and Education Network)
    • Cupertino, Kalifornien: HP
    192.6.38.127: ntp-cup.external.hp.com
    Servicebereich: USA Westküste
    • Newark, Delaware: Conectiv Communications
    138.39.7.20: ntp1.delmarva.com
    Servicebereich: Cable & Wireless Network (früher MCInet)
    • University Park, Pennsylvania: Penn state University
    128.118.46.3: otc1.psu.edu
    Servicebereich: NSFNET, PREPNET und JvNCnet

    Europa
    • Borowiec, Polen: Astrogeodynamical Observatory, Space Research Centre
    150.254.183.15: vega.cbk.poznan.pl
    Servicebereich: Polen und Europa
    • Stockholm, Schweden: Stupi AB
    192.36.143.151: Time2.Stupi.SE
    Servicebereich: Europa
    • Turin, Italien: IEN Galileo Ferraris
    193.204.114.1: time.ien.it
    Servicebereich: Italien und Europa
    • Zürich, Schweiz: Integrated Systems Laboratory , Eidgenössischen Technischen Hochschule Zürich
    129.132.2.21: swisstime.ethz.ch
    Servicebereich: Schweiz und Europa
    • Turin, Italien: CSTV of National Research Council
    150.145.33.1: tempo.cstv.to.cnr.it
    Servicebereich: Italien und Europa
    • Erlangen, Deutschland: Universität Erlangen-Nürnberg
    ntp0.fau.de; ntp1.fau.de; ntp2.fau.de;
    ntps1-0.uni-erlangen.de; ntps1-1.uni-erlangen.de; ntps1-2.uni-erlangen.de
    Servicebereich: Deutschland und Europa
    • Berlin, Deutschland: Technische Universität Berlin
    130.149.17.21: ntps1-0.cs.tu-berlin.de
    130.149.17.8: ntps1-1.cs.tu-berlin.de
    Servicebereich: Deutschland und Europa
    • Deutschland
    131.173.17.7: ntps1-1.rz.Uni-Osnabrueck.DE
    Servicebereich: Deutschland und Europa
    • Schweden
    192.36.143.150: Time1.Stupi.SE
    Servicebereich: SUnet und NORDUnet Schweden

    Fernost und pazifische Randgebiete
    • Hong Kong: Chinesische Universität von Hong Kong.
    137.189.6.18: clock.cuhk.edu.hk
    Servicebereich: Hong Kong (China) und Südostasien
    • Fukuoka, Japan: Universität Fukuoka
    133.100.9.2: clock.nc.fukuoka-u.ac.jp
    133.100.11.8: clock.tl.fukuoka-u.ac.jp
    Servicebereich: Japan und pazifischer Raum

    Australien
    • Melbourne, Australien: University of Melbourne
    128.250.36.2: ntp.cs.mu.OZ.AU
    Servicebereich: Australien und Neuseeland

    Zeitserver der zweiten Ebene
    Nach geographischem Standort sortiert:
    Nordamerika
    NTP-Zeitserver: • Quebec, Kanada: Canadian Meteorological Center
    ntp1.cmc.ec.gc.ca; ntp2.cmc.ec.gc.ca
    Servicebereich: Ostkanada
    • Ontario, Kanada: National Research Council of Canada
    time.chu.nrc.ca; time.nrc.ca
    Servicebereich: Kanada
    • Saskatchewan, Kanada: University of Regina
    142.3.100.15: timelord.uregina.ca
    Servicebereich: Kanada
    • Ontario, Kanada: University of Toronto
    tick.utoronto.ca; tock.utoronto.ca
    Servicebereich: Ostkanada
    • Mexiko: Audiotel-Büro
    ntp2a.audiotel.com.mx; ntp2c.audiotel.com.mx; ntp2b.audiotel.com.mx
    Servicebereich: Avantel, MCINet und Mexiko
    • Santa Cruz, Kalifornien: Scruz-net, inc.
    165.227.1.1: ns.scruz.net
    Servicebereich: Westen der USA
    • San Diego, Kalifornien: UCSD Academic Computing Services/Network Operations
    132.239.254.49: ntp.ucsd.edu
    Servicebereich: CERFNET; NSFNET, SDSC-Bereich, und nahegelegene Bereiche
    • Quincy, Kalifornien
    ntp1.mainecoon.com; ntp2.mainecoon.com
    Servicebereich: Nordamerika
    • Newark, Delaware: University of Delaware
    128.175.1.3: louie.udel.edu
    Servicebereich: CAIRN, Abilene und vBNS
    • Atlanta, Georgia: CNSG
    ntp.shorty.com
    Servicebereich: Südwesten der USA
    • Kennesaw, Georgia: PeachNet
    rolex.peachnet.edu; timex.peachnet.edu
    Servicebereich: PeachNet (Georgia) und Südwesten der USA
    • Urbana-Champaign, Illinois: University of Illinois
    ntp-0.cso.uiuc.edu; ntp-1.cso.uiuc.edu; ntp-2.cso.uiuc.edu
    Servicebereich: CICNET, Mittlerer Westen und NCSA-Bereich
    • Chicago, Illinois: Argonne National Laboratory
    ntp-1.mcs.anl.gov; ntp-2.mcs.anl.gov
    Servicebereich: NSF/ANSNet, CICNet, NetIllinois und ESNet
    • West Lafayette, Indiana: Purdue University
    gilbreth.ecn.purdue.edu; harbor.ecn.purdue.edu; molecule.ecn.purdue.edu
    Servicebereich: NSFNET- und CICNET-Bereich
    • Manhattan, Kansas: KansasNet OnLine Services
    199.240.130.1: ntp1.kansas.net
    199.240.130.12: ntp2.kansas.net
    Servicebereich: Zentral-USA und Great Plains
    • Boston, Massachusetts: UMass-Boston CS dept.
    158.121.104.4: timeserver.cs.umb.edu
    Servicebereich: Neuengland
    • Minneapolis/St Paul, Minnesota: University of Minnesota
    ns.nts.umn.edu; nss.nts.umn.edu
    Servicebereich: CICNET-Bereich
    • Columbia, Missouri: University of Missouri-Columbia
    128.206.206.12: everest.cclabs.missouri.edu
    Servicebereich: MOREnet
    • Omaha, Nebraska: Radiks Internet Access
    205.138.126.83: allison.radiks.net
    Servicebereich: Mittlerer Westen, USA
    • Las Vegas, Nevada: University of Nevada System Computing Services
    131.216.1.101: cuckoo.nevada.edu
    Servicebereich: NevadaNet, NSFNET und SDSC-Bereich
    • Las Vegas, Nevada: UNLV College of Engineering
    tick.cs.unlv.edu; tock.cs.unlv.edu
    Servicebereich: Sprintnet
    • New York City, New York: Columbia University
    ntp.ctr.columbia.edu
    Servicebereich: Sprintlink und NYSERnet
    • Ithaca, New York: Cornell University
    192.35.82.50: ntp0.cornell.edu
    Servicebereich: NSFNET und NYSER-Bereich
    • New York, New York: Morningside Campus, Columbia University
    sundial.columbia.edu
    Servicebereich: NYSERnet
    • New York City, New York: Columbia University Computer Science Department
    timex.cs.columbia.edu
    Servicebereich: PSINET; NSFNET, und NYSER-Bereich
    • Norman, Oklahoma: University of Oklahoma
    129.15.22.8: constellation.ecn.uoknor.edu
    Servicebereich: Midnet
    • Coos Bay, Oregon: Koala Computers
    207.48.109.6: tick.koalas.com
    Servicebereich: Nordwesten der USA
    • University Park, Pennsylvania: Penn state University
    128.118.25.3: clock.psu.edu
    Servicebereich: Internet2, vBNS, CERFnet(AT&T IP Services), PSC/NCNE und CASC
    • Pittsburgh, Pennsylvania: Pittsburgh Supercomputing Center
    128.182.58.100: fuzz.psc.edu
    Servicebereich: NSFNET und PSC-Bereich
    • Pittsburgh, Pennsylvania: Carnegie Mellon Electrical and Computer Engineering
    ntp-1.ece.cmu.edu; ntp-2.ece.cmu.edu
    Servicebereich: PREPNET und PSC-Bereich
    • Dallas, Texas: Cox School of Business, Southern Methodist University
    129.119.80.126: ntp.cox.smu.edu
    Servicebereich: NSFNET und SESQUI-Bereich
    • Hughes Springs, Texas: First National Bank
    209.144.20.76: ntp.fnbhs.com
    Servicebereich: Nordosten Texas
    • Houston, Texas: Baylor College of Medicine
    128.249.1.10: ntp.tmc.edu
    Servicebereich: NSFNET und SESQUI-Bereich
    • College Station, Texas: Texas A&M University
    165.91.52.110: ntp5.tamu.edu
    Servicebereich: NSFNET, SESQUI-Bereich, THEnet und TAMUSDSN
    • Plano, Texas: Greyware Automation Products
    tick.greyware.com; tock.greyware.com
    Servicebereich: Südzentral-USA
    • Blacksburg, Virginia: Virginia Tech Computing Center
    ntp-1.vt.edu; ntp-2.vt.edu
    Servicebereich: Südwesten der USA
    • Arlington, Virginia: Center for Seismic Studies
    140.162.1.3: ntp.cmr.gov
    Servicebereich: NSFNET und SURA-Bereich
    • Richland, Washington: Washington state University
    192.31.216.30: clock.tricity.wsu.edu
    Servicebereich: NSFNET und NorthWestNet
    • Washington, USA: Mill Creek
    time.ultimeth.net
    Servicebereich: Nordwesten der USA
    • Wisconsin, USA: Computer Science Department, University of Wisconsin-Madison
    ntp1.cs.wisc.edu; ntp2.cs.wisc.edu; ntp3.cs.wisc.edu
    Servicebereich: USA und jeder andere

    Südamerika
    • Buenos Aires, Argentinien: Network Access Point
    200.49.40.1: CNAME: tick.nap.com.ar
    200.49.32.1: CNAME: tock.nap.com.ar
    Servicebereich: Argentinien
    • Buenos Aires, Argentinien: Sinectis S.A.
    time.sinectis.com.ar
    Servicebereich: Argentinien
    • Brasilien: Brazilian Research Network
    200.144.121.33: ntp.cais.rnp.br
    Servicebereich: Brasilien
    • Venezuela: VELUG, Grupo de Usuarios Linux de Venezuela
    150.185.192.250: ntp.linux.org.ve
    Servicebereich: Arica

    Europa
    • Zürich, Schweiz: Eidgenössischen Technischen Hochschule Zürich
    129.132.98.11: bernina.ethz.ch
    Servicebereich: Schweiz und Europa
    • Standort: Kopenhagen, Dänemark, Europa
    clock.netcetera.dk; clock2.netcetera.dk
    Servicebereich: Dänemark, Skandinavien und Nordeuropa
    • Spanien: Altea
    slug.ctv.es
    Servicebereich: Spanien
    • Pieksamaki, Finnland: Keski-Savon Oppimiskeskus
    tick.keso.fi; tock.keso.fi
    Servicebereich: Finnland
    • Meudon, Frankreich: Observatoire de Paris-Meudon
    ntp.obspm.fr
    Servicebereich: Frankreich und Europa
    • Lyon, Frankreich: CISM
    ntp.univ-lyon1.fr
    Servicebereich: Frankreich, Schweiz, Italien und Europa
    • Paris, Frankreich: VIA, Ecole Centrale
    138.195.130.70: ntp.via.ecp.fr
    Servicebereich: Frankreich und Europa
    • Budapest, Ungarn: KFKI Research Institute for Particle and Nuclear Physics
    148.6.0.1: time.kfki.hu
    Servicebereich: HUNGARNET
    • Italien: Net4u Srl, Vercelli, Italien
    195.32.52.129: ntps.net4u.it
    Servicebereich: Italien
    • Oslo, Norwegen: Universität Oslo
    129.240.64.3: fartein.ifi.uio.no
    Servicebereich: NORDUnet
    • Oslo, Norwegen: Alcanet International
    time.alcanet.no
    Servicebereich: Europa
    • Krakau, Polen: Academic Computer Centre
    149.156.4.11: info.cyf-kr.edu.pl
    Servicebereich: Polen und Europa
    • Lund, Schweden: Lund Institute of Technology
    130.235.20.3: ntp.lth.se
    Servicebereich: Schweden und NORDUnet
    • Ljubljana, Slowenien: Institute of Biophysics, University of Ljubljana
    biofiz.mf.uni-lj.si 193.2.69.11
    Servicebereich: Slowenien und Europa
    • Ljubljana, Slowenien: Hydrometeorological Institute of Slovenia
    hmljhp.rzs-hm.si
    Servicebereich: Slowenien und Europa
    • Ljubljana, Slowenien: Academic and Research Network of Slovenia
    ntp1.arnes.si; ntp2.arnes.si
    Servicebereich: Slowenien und Europa
    • Ljubljana, Slowenien: J. Stefan Institute
    time.ijs.si
    Servicebereich: Slowenien und Europa

    Britische Inseln
    • Dublin, Irland: School of Mathematics, Trinity College
    ntp.cs.tcd.ie; ntp.maths.tcd.ie; ntp.tcd.ie
    Servicebereich: Irland und Großbritannien
    • Glasgow, Schottland: Strathclyde University
    ntp.cs.strath.ac.uk
    Servicebereich: Großbritannien, Europa und andere
    • Cambridge, Großbritannien
    ntp0.uk.uu.net; ntp1.uk.uu.net;
    ntp2.uk.uu.net
    Servicebereich: UUNET (in Großbritannien früher auch als PIPEX bekannt) und Großbritannien.
    • Manchester, England: University of Manchester
    ntp2a.mcc.ac.uk; ntp2b.mcc.ac.uk;
    ntp2c.mcc.ac.uk; ntp2d.mcc.ac.uk
    Servicebereich: Großbritannien
    • Buckinghamshire, Großbritannien: Wibble U.K., Aylesbury
    tick.tanac.net
    Servicebereich: Großbritannien

    Asien
    • Moskau, Russland: Landau Institute for Theoretical Physics
    193.233.9.7: ntp.landau.ac.ru
    Servicebereich: Russland
    • Russland: Pushchino (bei Moskau)
    194.149.67.130: ntp.psn.ru
    Servicebereich: Russland
    • Chernogolovka, Russland: Chernogolovka Scientific Center (bei Moskau)
    193.233.46.10: sign.chg.ru
    Servicebereich: Russland

    Fernost und pazifische Randgebiete
    • Tokyo, Japan: Cyber Fleet, Inc.
    203.139.30.195: ntp.cyber-fleet.net
    Servicebereich: Japan und Ostasien
    • Seoul, Korea: Inet, Inc.
    time.nuri.net
    Servicebereich: Korea, Japan, Hong Kong und Ostasien
    • Hamilton, Neuseeland: Universität Waikato
    truechimer.waikato.ac.nz; truechimer1.waikato.ac.nz;
    truechimer2.waikato.ac.nz; truechimer3.waikato.ac.nz
    Servicebereich: Neuseeland
    • Singapur und Philippinen:
    ntp.shim.org
    Servicebereich: Singapur

    Afrika
    • Lagos, Nigeria: Supernet300
    ntp.supernet300.com
    Servicebereich: Westafrika (hauptsächlich nigerischer NITEL-Backbone)
    • Pietermaritzburg, Südafrika: Natal University
    143.128.82.200: ntp.cs.unp.ac.za
    Servicebereich: Südafrika

    Australien
    • Adelaide, Südaustralien: University of Adelaide
    129.127.28.4: augean.eleceng.adelaide.edu.au
    129.127.40.3: ntp.adelaide.edu.au
    203.21.37.18: ntp.saard.net
    Servicebereich: AARNet
    • Carlton, Victoria, Australien: eSec Limited
    203.21.84.4: time.esec.com.au

    *)
END_FUNCTION_BLOCK

(* ---- SNTP_SERVER.st ---- *)
FUNCTION_BLOCK SNTP_SERVER
    (*http://www.oscat.de/images/OSCATNetwork/oscat_netlib121_en.pdf#page=128*)
    (* Domain Name System (query) *)
    tx := T_PLC_MS(); (* read system time *)

    CASE state OF

    00: (* Warten auf Freigabe *)
    	IF ENABLE THEN
    		state := 10;
    		ip_state := BYTE#1; (* Anmelden *)
        		(*####################  DEBUG-MESSAGE  ###################################*)
        		(*IF _debug_enable THEN
          			LOG_CL.NEW_MSG := 'SNTP_SERVER: S00 START';
          			LOG_MSG();
        		END_IF*)
        		(*########################################################################*)
    	END_IF

    10: (* Bei IP_Control anmelden und auf freigabe warten *)
    	IF ip_state = BYTE#3 THEN
    		(* IP Datenverkehr einrichten *)
    		IP_C.C_PORT := WORD#123; (* Portnummer eintragen *)
    		IP_C.C_IP := DWORD#00; (* IP eintragen *)
    		IP_C.C_MODE := BYTE#5; (* Mode: UDP+PASSIV+PORT *)
    		IP_C.C_ENABLE := TRUE; (* Verbindungsaufbau freigeben *)
    		IP_C.TIME_RESET := TRUE; (* Zeitueberwachung rücksetzen *)
    		IP_C.R_OBSERVE := FALSE; (* Datenempfang ueberwachen *)
    		S_BUF.SIZE := UINT#0; (* Sendelänge eintragen *)
    		R_BUF.SIZE := UINT#0; (* Empfangslänge rücksetzen *)
    		state := 20;
        		(*####################  DEBUG-MESSAGE  ###################################*)
        		(*IF _debug_enable THEN
          			LOG_CL.NEW_MSG := 'SNTP_SERVER: S10 INIT';
          			LOG_MSG();
        		END_IF*)
        		(*########################################################################*)
    	END_IF
    20:
    	IF R_BUF.SIZE > UINT#0 THEN
    		state := 20;
        		(*####################  DEBUG-MESSAGE  ###################################*)
        		(*IF _debug_enable THEN
          			LOG_CL.NEW_MSG := 'SNTP_SERVER: S20 REQUEST - Size: ~1';
          			LOG_CL.PRINTF[1] := UINT_TO_STRING(R_BUF.SIZE);
          			LOG_MSG();
        		END_IF*)
        		(*########################################################################*)
    		(* empfangenes Telegramm mit 00 auffüllen , wenn zu kurz ! und Sendebuffer mit 00 vorbelegen *)
    		FOR i := 0 TO 47 DO
    			IF INT_TO_UINT(i) > R_BUF.SIZE - 1 THEN
    				R_BUF.BUFFER[i] := BYTE#00;
    			END_IF
    			S_BUF.BUFFER[i] := BYTE#00;
    		END_FOR

    		R_BUF.SIZE := UINT#0;

    		(* Sendedaten aufbereiten *)
    		S_BUF.BUFFER[0] := BYTE#2#11100; (* Flags: NO WARNING, NTP VERSION 3 , SERVER *)
    		S_BUF.BUFFER[1] := STRATUM; (* Peer Clock STRATUM: *)
    		S_BUF.BUFFER[2] := BYTE#10; (* Peer Polling Intervall 2 hoch 10 = 1024 sek. *)
    		S_BUF.BUFFER[3] := BYTE#16#FB; (* Peer Clock Precision: -5 = -31,25ms *)

    		(* Umrechnung SNTP Timestamp Base 1900-01-01 = Unix 1970-01-01 + 2208988800 sekunden *)
    		timestamp_int := DT_TO_DWORD(UDT) + DWORD#2208988800;

    		(* Sekundenanteile sind als 32 Bit Fractal dargestellt *)
    		(* nur mit veringerte Auflösung berechnen 1/65535 -> Highword verwenden *)
    		(* Berechnung des Sekundenanteils: XMS * 65535 / 1000 *)
    		timestamp_sek := DINT_TO_DWORD(DWORD_TO_DINT(SHL(INT_TO_DWORD(XMS),16))/DINT#1000);

    		ts_b := BYTE_OF_DWORD(timestamp_int,3); (* Timestamp Byte 3 *)
    		S_BUF.BUFFER[16] := ts_b; (* Reference Timestamp *)
    		S_BUF.BUFFER[32] := ts_b; (* Receive   Timestamp *)
    		S_BUF.BUFFER[40] := ts_b; (* Transmit  Timestamp *)

    		ts_b := BYTE_OF_DWORD(timestamp_int,2); (* Timestamp Byte 2 *)
    		S_BUF.BUFFER[17] := ts_b; (* Reference Timestamp *)
    		S_BUF.BUFFER[33] := ts_b; (* Receive   Timestamp *)
    		S_BUF.BUFFER[41] := ts_b; (* Transmit  Timestamp *)

    		ts_b := BYTE_OF_DWORD(timestamp_int,1); (* Timestamp Byte 1 *)
    		S_BUF.BUFFER[18] := ts_b; (* Reference Timestamp *)
    		S_BUF.BUFFER[34] := ts_b; (* Receive   Timestamp *)
    		S_BUF.BUFFER[42] := ts_b; (* Transmit  Timestamp *)

    		ts_b := BYTE_OF_DWORD(timestamp_int,0); (* Timestamp Byte 0 *)
    		S_BUF.BUFFER[19] := ts_b; (* Reference Timestamp *)
    		S_BUF.BUFFER[35] := ts_b; (* Receive   Timestamp *)
    		S_BUF.BUFFER[43] := ts_b; (* Transmit  Timestamp *)

    		ts_b := BYTE_OF_DWORD(timestamp_sek,1); (* Timestamp Byte 1 *)
    		S_BUF.BUFFER[20] := ts_b; (* Reference Timestamp *)
    		S_BUF.BUFFER[36] := ts_b; (* Receive   Timestamp *)
    		S_BUF.BUFFER[44] := ts_b; (* Transmit  Timestamp *)

    		ts_b := BYTE_OF_DWORD(timestamp_sek,0);	(* Timestamp Byte 0 *)
    		S_BUF.BUFFER[21] := ts_b; (* Reference Timestamp *)
    		S_BUF.BUFFER[37] := ts_b; (* Receive   Timestamp *)
    		S_BUF.BUFFER[45] := ts_b; (* Transmit  Timestamp *)

    		(* Byte 1-8 von Transmit-Time auf Originate-Time umkopieren *)
    		i2 := 40;
    		FOR i := 24 TO 31 DO
    			S_BUF.BUFFER[i] := R_BUF.BUFFER[i2];
    			i2 := i2 +1;
    		END_FOR

    		S_BUF.SIZE := UINT#48; (* Daten senden *)

    	ELSIF NOT ENABLE AND S_BUF.SIZE = UINT#0 THEN
    		ip_state := BYTE#4; (* Abmelden *)
    		state := 0;
    	END_IF

    END_CASE

    t(IN:= IP_C.ERROR > DWORD#0, PT:=t#5s);
    IF t.Q THEN
      IP_C.TIME_RESET := TRUE; (* Error Reset *)
    END_IF

    (* IP_FIFO *)
    IP_FIFO(FIFO:=IP_C.FIFO,state:=ip_state,ID:=ip_id);

    (* revision history
    ks	18. oct. 2008	rev 1.0
    	original version

    ks	20. oct. 2009	rev 1.1
    	Networkbuffer und Buffer-funktionen auf Basis 0

    ks	17. may. 2011	rev 1.2
    	automatischer re-connect
    *)

    (*               SNTP(NTP) Datenstruktur
                                      1                   2                   3
                  0 1 2 3 4 5 6 7 8 9 0 1 2 3 4 5 6 7 8 9 0 1 2 3 4 5 6 7 8 9 0 1
                 +-+-+-+-+-+-+-+-+-+-+-+-+-+-+-+-+-+-+-+-+-+-+-+-+-+-+-+-+-+-+-+-+
    Byte: 01-04  |LI | VN  |Mode |    STRATUM    |     Poll      |   Precision   |
                 +-+-+-+-+-+-+-+-+-+-+-+-+-+-+-+-+-+-+-+-+-+-+-+-+-+-+-+-+-+-+-+-+
    Byte: 05-08  |                          Root  Delay (32 Bit)                 |
                 +-+-+-+-+-+-+-+-+-+-+-+-+-+-+-+-+-+-+-+-+-+-+-+-+-+-+-+-+-+-+-+-+
    Byte: 09-12  |                       Root  Dispersion (32 Bit)               |
                 +-+-+-+-+-+-+-+-+-+-+-+-+-+-+-+-+-+-+-+-+-+-+-+-+-+-+-+-+-+-+-+-+
    Byte: 13-16  |                     Reference Identifier (32 Bit)             |
                 +-+-+-+-+-+-+-+-+-+-+-+-+-+-+-+-+-+-+-+-+-+-+-+-+-+-+-+-+-+-+-+-+
    Byte: 17-24  |                    Reference Timestamp (64 Bit)               |
                 +-+-+-+-+-+-+-+-+-+-+-+-+-+-+-+-+-+-+-+-+-+-+-+-+-+-+-+-+-+-+-+-+
    Byte: 25-32  |                    Originate Timestamp (64 Bit)               |
                 +-+-+-+-+-+-+-+-+-+-+-+-+-+-+-+-+-+-+-+-+-+-+-+-+-+-+-+-+-+-+-+-+
    Byte: 33-40  |                     Receive Timestamp (64 Bit)                |
                 +-+-+-+-+-+-+-+-+-+-+-+-+-+-+-+-+-+-+-+-+-+-+-+-+-+-+-+-+-+-+-+-+
    Byte: 41-48  |                     Transmit Timestamp (64 Bit)               |
                 +-+-+-+-+-+-+-+-+-+-+-+-+-+-+-+-+-+-+-+-+-+-+-+-+-+-+-+-+-+-+-+-+
    Byte: 49-52  |                 Key Identifier (optional) (32 Bit)            |
                 +-+-+-+-+-+-+-+-+-+-+-+-+-+-+-+-+-+-+-+-+-+-+-+-+-+-+-+-+-+-+-+-+
    Byte: 53-68  |                 Message Digest (optional) (128 Bit)           |
                 +-+-+-+-+-+-+-+-+-+-+-+-+-+-+-+-+-+-+-+-+-+-+-+-+-+-+-+-+-+-+-+-+
    *)
END_FUNCTION_BLOCK

(* ---- SPIDER_ACCESS.st ---- *)
FUNCTION_BLOCK SPIDER_ACCESS
    (*http://www.oscat.de/images/OSCATNetwork/oscat_netlib121_en.pdf#page=129*)
    CASE state OF

    00:
    	IF MODE > BYTE#0 AND MODE < BYTE#3 THEN
    		mode_save := MODE; (* Modus speichern *)
    		(* wenn kein '.' in Name dann ist es eine globale variable *)
    		IF FIND(VAR_NAME,'.') = 0 THEN
    			st_tmp := CONCAT('%40GV.',VAR_NAME);
    		ELSE
    			st_tmp := VAR_NAME;
    		END_IF

    		IF mode_save = BYTE#2 THEN (* 2 = Write *)
    			value_len := INT_TO_UINT(LEN(VALUE));
    			st_tmp := CONCAT(st_tmp,'+');
    			st_tmp := CONCAT(st_tmp,VALUE);
    			URL_DATA:=STRING_TO_URL(STR:= CONCAT('http://x/dir/cgi-bin/writeVal.exe?',st_tmp),DEFAULT_PROTOCOL:='',DEFAULT_PATH:='');
    		ELSE
    			URL_DATA:=STRING_TO_URL(STR:= CONCAT('http://x/dir/cgi-bin/readVal.exe?',st_tmp),DEFAULT_PROTOCOL:='',DEFAULT_PATH:='');
    		END_IF

    		state := 60;
    	END_IF
    60:
    	IF HTTP_GET.DONE THEN
    		IF mode_save = BYTE#2 THEN (* Write *)
    			body_len := HTTP_GET.BODY_STOP - HTTP_GET.BODY_START + BOOL_TO_UINT(HTTP_GET.BODY_STOP > UINT#0);
    			ERROR := BOOL_TO_DWORD(body_len <> value_len);
    		ELSE (* Read *)
    			IF HTTP_GET.BODY_START > 0 THEN
    				VALUE := BUFFER_TO_STRING(PT:=ADR(R_BUF.BUFFER),SIZE:=R_BUF.SIZE,START:=UINT_TO_INT(HTTP_GET.BODY_START),STOP:=UINT_TO_INT(HTTP_GET.BODY_STOP));
    			ELSE
    				VALUE := '';
    			END_IF
    		END_IF
    		state   := 100;

    	ELSIF (HTTP_GET.ERROR > DWORD#00) THEN
    		ERROR := HTTP_GET.ERROR;
    		state   := 100;
    	END_IF

    100:
    	(* UNLOCK HTTP DATA *)
    	IF HTTP_GET.DONE = FALSE THEN
    		state := 0;
    	END_IF

    END_CASE

    (* HTTP_GET *)
    HTTP_GET(	IP_C:=IP_C,
    			S_BUF:=S_BUF,
    			R_BUF:=R_BUF,
    			IP4:=DWORD#00,
    			GET:=state=60,
    			MODE:=BYTE#0,
    			UNLOCK_BUF:=state=100,
    			URL_DATA:=URL_DATA
    			);

    (* revision history
    ks	18. mar. 2009	rev 1.0
    	original version

    ks	12. apr. 2011	rev 1.1
    	fehlerkorrektur bei buffer_to_string
    *)
END_FUNCTION_BLOCK

(* ---- SYS_LOG.st ---- *)
FUNCTION_BLOCK SYS_LOG
    (*http://www.oscat.de/images/OSCATNetwork/oscat_netlib121_en.pdf#page=131*)
    CASE state OF
    00: (* auf positive Flanke SET warten *)
    	IF ACTIVATE AND NOT activate_last THEN
    		state := 10;
    		ERROR := DWORD#0;
    		ip_state := BYTE#1; (* Anmelden *)
        		(*####################  DEBUG-MESSAGE  ###################################*)
        		(*IF _debug_enable THEN
          			LOG_CL.NEW_MSG := 'SYS_LOG: S00 START /ip_id ~4';
          			LOG_CL.PRINTF[4]  := BYTE_TO_STRING(ip_id);
          			LOG_MSG();
        		END_IF*)
        		(*########################################################################*)
    	END_IF
    	DONE_P := FALSE;

    10: (* Bei IP_Control anmelden und auf freigabe warten *)
    	IF ip_state = BYTE#3 THEN
    		(* Sendedaten aufbereiten *)
    		i := 0;
    		IF (OPTION AND BYTE#0000_0001) = BYTE#00 THEN (* OPTION: no priority Code *)
    			(* Priority:  '<xx>' als dezimalwert *)
    			(* BYTE: xxxx x...  = FACILITY *)
    			(*       .... .xxx  = Level *)
    			s1 := REPLACE('<P>',BYTE_TO_STRING(SHL(FACILITY,3) OR (SEVERITY AND BYTE#0000_0111)),1,2);
    		ELSE
    			s1 := '';
    		END_IF

    		IF (OPTION AND BYTE#0000_0010) = BYTE#00 THEN (* OPTION: No Use Syslog RFC Header *)
    			(* 'month day hh:mm:ss ' *)
    			s1 := CONCAT(s1,DT_TO_STRF(DTI:=LOC_DT,MS:=0,FMT:='#E #W #N:#R:#T ',LANG:=1));
    			_STRING_TO_BUFFER(STR:=s1,POS:=i,PT:=ADR(S_BUF.BUFFER),SIZE:=UINT#1024);
    			i := i + LEN(s1);
    			(* ' sourcename eintragen *)
    			_STRING_TO_BUFFER(STR:=HOSTNAME,POS:=i,PT:=ADR(S_BUF.BUFFER),SIZE:=UINT#1024);
    			i := i + LEN(HOSTNAME);
    			S_BUF.BUFFER[i] := BYTE#32; (* leerzeichen einfuegen *)
    			i := i + 1;
    			(* ' TAG eintragen *)
    			_STRING_TO_BUFFER(STR:=TAG,POS:=i,PT:=ADR(S_BUF.BUFFER),SIZE:=UINT#1024);
    			i := i + LEN(TAG);
    			S_BUF.BUFFER[i] := BYTE#32; (* leerzeichen einfuegen *)
    			i := i + 1;
    		END_IF

    		(* ' MESSAGE eintragen *)
    		_STRING_TO_BUFFER(STR:=MESSAGE,POS:=i,PT:=ADR(S_BUF.BUFFER),SIZE:=UINT#1024);
    		i := i + LEN(MESSAGE);

    		IF (OPTION AND BYTE#0000_0100) > BYTE#00 THEN (* OPTION: Add a CR & LF to end of MESSAGE *)
    			S_BUF.BUFFER[i] := BYTE#13; (* Carriage Return einfuegen *)
    			i := i + 1;
    			S_BUF.BUFFER[i] := BYTE#10; (* Linefeed einfuegen *)
    			i := i + 1;
    		END_IF

    		state := 30;

    		(* IP Datenverkehr einrichten *)
    		IF (OPTION AND BYTE#2#0000_1000) > BYTE#00 THEN (* OPTION: TCP Mode *)
    			IP_C.C_MODE := BYTE#0; (* Mode: TCP/AKTIV *)
    		ELSE
    			IP_C.C_MODE := BYTE#1; (* Mode: UDP/AKTIV *)
    		END_IF

    		IF PORT = WORD#0 THEN (* keine Portnummer vorgegeben ? *)
    			IF IP_C.C_MODE = BYTE#0 THEN (* Modus bestimmen  TCP oder UDP ? *)
    				IP_C.C_PORT := WORD#1468; (* Standard Portnummer für Syslog over TCP *)
    			ELSE
    				IP_C.C_PORT := WORD#514; (* Standard Portnummer für Syslog over UDP *)
    			END_IF
    		ELSE
    			IP_C.C_PORT := PORT; (* uebergebene Portnummer eintragen *)
    		END_IF

    		IP_C.C_IP := SERVER_IP4; (* IP eintragen *)
    		IP_C.C_ENABLE := TRUE; (* Verbindungsaufbau freigeben *)
    		IP_C.TIME_RESET := TRUE; (* Zeitueberwachung rücksetzen *)
    		IP_C.R_OBSERVE := FALSE; (* Datenempfang ueberwachen *)
    		S_BUF.SIZE := INT_TO_UINT(i); (* Sendelänge eintragen *)
    		R_BUF.SIZE := UINT#0; (* Empfangslänge rücksetzen *)
        		(*####################  DEBUG-MESSAGE  ###################################*)
        		(*IF _debug_enable THEN
          			LOG_CL.NEW_MSG := 'SYS_LOG: S20 SEND /ip_id ~4';
          			LOG_CL.PRINTF[4]  := BYTE_TO_STRING(ip_id);
          			LOG_MSG();
        		END_IF*)
        		(*########################################################################*)
    	END_IF

    30:
    	IF IP_C.ERROR <> DWORD#00 THEN
    		ERROR := IP_C.ERROR;
    		state := 0;
        		(*####################  DEBUG-MESSAGE  ###################################*)
        		(*IF _debug_enable THEN
          			LOG_CL.NEW_MSG := 'SYS_LOG: S30 ERROR ~1 ip_id ~4';
          			LOG_CL.PRINTF[1]  := DWORD_TO_STRING(ERROR);
          			LOG_CL.PRINTF[4]  := BYTE_TO_STRING(ip_id);
          			LOG_MSG();
        		END_IF*)
        		(*########################################################################*)
    	ELSIF S_BUF.SIZE = UINT#0 THEN (* warten bis alle daten gesendet sind *)
    		DONE_P := TRUE;
    		state := 0;
        		(*####################  DEBUG-MESSAGE  ###################################*)
        		(*IF _debug_enable THEN
          			LOG_CL.NEW_MSG := 'SYS_LOG: S30 OK /ip_id ~4';
          			LOG_CL.PRINTF[4]  := BYTE_TO_STRING(ip_id);
          			LOG_MSG();
        		END_IF*)
        		(*########################################################################*)
    	END_IF

    	IF state = 0 THEN (* Verbindung freigeben *)
    		ip_state := BYTE#4;
    	END_IF

    END_CASE

    activate_last := ACTIVATE; (* letzten Status sichern zur Flankenerkennung *)

    (* IP_FIFO *)
    IP_FIFO(FIFO:=IP_C.FIFO,state:=ip_state,ID:=ip_id);

    (* revision history
    ks	18. oct. 2008	rev 1.0
    	original version

    ks	20. jun. 2009	rev 1.1
    	Networkbuffer und Buffer-funktionen auf Basis 0

    *)
END_FUNCTION_BLOCK

(* ---- TELNET_LOG.st ---- *)
FUNCTION_BLOCK TELNET_LOG
    (*http://www.oscat.de/images/OSCATNetwork/oscat_netlib121_en.pdf#page=135*)
    IF NOT init THEN
    	init := TRUE;
    	IF OPTION > 0 THEN
    		TELNET_PRINT.OPTION := OPTION;
    	END_IF
    	IF PORT > 0 THEN (* bei portvorgabe wird der standardport überschrieben *)
    		TELNET_PRINT.PORT := PORT;
    	END_IF
      	watchdog.PT := T#1ms;
    END_IF

    watchdog(IN:=FALSE); (* Timer stoppen *)

    ci := LOG_CL.IDX;

    (* CONNECT_OFF Flanke auswerten *)
    IF IP_C.C_STATE = BYTE#1 THEN
    	pi := 0;
    	init := FALSE;
    END_IF

    REPEAT
    	IF pi <> ci AND IP_C.C_STATE > BYTE#127 THEN
    		IF pi = 0 AND LOG_CL.RING_MODE THEN pi := ci; END_IF
    		pi_last := pi;
    		pi := pi + 1;
    		IF pi > LOG_CL.SIZE THEN pi := 1; END_IF
    		send := TRUE;
    	ELSE
    		send := FALSE;
    	END_IF

    	TELNET_PRINT(	IP_C := IP_C,
    					S_BUF := S_BUF,
    					ENABLE := ENABLE,
    					send := send,
    					TEXT := LOG_CL.MSG[pi],
    					BACK_COLOR := DWORD_TO_BYTE(SHL(LOG_CL.MSG_OPTION[pi],8)),
    					FRONT_COLOR := DWORD_TO_BYTE(LOG_CL.MSG_OPTION[pi] ));
    	READY := TELNET_PRINT.READY;
    	done := TELNET_PRINT.done;

    	IF send AND NOT done THEN
    		pi := pi_last;
    	END_IF

    	watchdog(IN:=TRUE);

    UNTIL (watchdog.Q OR NOT done )
    END_REPEAT

    (* revision history
    ks	14. aug. 2009	rev 1.0
    	original version

    ks	03. dec. 2011	rev 1.1
    	neue parameter und initialisierung optimiert

    *)
END_FUNCTION_BLOCK

(* ---- TELNET_PRINT.st ---- *)
FUNCTION_BLOCK TELNET_PRINT
    (*http://www.oscat.de/images/OSCATNetwork/oscat_netlib121_en.pdf#page=137*)
    READY := IP_C.C_STATE > BYTE#127;
    DONE := FALSE;

    CASE state OF

    00: (* Warten auf Freigabe *)
    	IF ENABLE THEN
    		state := 10;
    		ip_state := BYTE#1; (* Anmelden *)
    	END_IF

    10: (* Bei IP_Control anmelden und auf freigabe warten *)
    	IF ip_state = BYTE#3 THEN

    		(* IP Datenverkehr einrichten *)
    		IP_C.C_PORT := PORT; (* Portnummer eintragen *)
    		IP_C.C_IP := DWORD#00; (* IP eintragen *)
    		IP_C.C_MODE := BYTE#4; (* Mode: TCP+PASSIV+PORT *)
    		IP_C.TIME_RESET := TRUE; (* Zeitueberwachung rücksetzen *)
    		IP_C.C_ENABLE := TRUE; (* Verbindungsaufbau freigeben *)
    		IP_C.R_OBSERVE := FALSE; (* keine Empfangsueberwachung *)
    		state := 20;
    	END_IF

    20:	IF IP_C.ERROR > DWORD#0 THEN
    		IP_C.TIME_RESET := TRUE; (* Fehler rücksetzen *)
    	END_IF
    	IF S_BUF.SIZE = UINT#0 THEN (* Datensenden nicht aktiv *)
    		IF NOT ENABLE THEN
    			ip_state := BYTE#4; (* Verbindung abbauen - Ressource freigeben *)
    			IP_C.C_ENABLE := FALSE; (* Verbindungsabbau *)
    			state := 0;
    		END_IF
    		IF IP_C.C_STATE = BYTE#1 THEN (* positive Flanke Connect off *)
    			init := FALSE;
    		ELSIF READY THEN (* Verbindung vorhanden *)
    			IF IP_C.C_STATE = BYTE#254 AND NOT init THEN (* positive Flanke Connect on *)
    				(* Var init ist notwendig, damit der Baustein im selben zyklus mehrmals ausgerufen werden kann *)
    				init := TRUE;
    				b0_screen_clear := (OPTION AND BYTE#2#0000_0001) > BYTE#0;
    				b1_autowrap := (OPTION AND BYTE#2#0000_0010) > BYTE#0;
    				b2_color := (OPTION AND BYTE#2#0000_0100) > BYTE#0;
    				b3_cr_lr := (OPTION AND BYTE#2#0000_1000) > BYTE#0;
    				b7_no_flush := (OPTION AND BYTE#2#1000_0000) > BYTE#0;

    				last_fc := NOT FRONT_COLOR; (* aktualisierung der Farben erzwingen !*)
    				x := 0;

    				(* AUTOWRAP OFF/ON *)
    				S_BUF.BUFFER[x] := BYTE#16#1B; (* ESC *)
    				x := x +1;
    				S_BUF.BUFFER[x] := BYTE#16#5B; (* [ *)
    				x := x +1;
    				S_BUF.BUFFER[x] := BYTE#16#3F; (* ? *)
    				x := x +1;
    				S_BUF.BUFFER[x] := BYTE#16#37; (* 7 *)
    				x := x +1;
    				S_BUF.BUFFER[x] := SEL(b1_autowrap, BYTE#16#6C (* l *),BYTE#16#68 (* h *));

    				IF b0_screen_clear THEN
    					IF b2_color THEN
    						x := x +1;
    						S_BUF.BUFFER[x] := BYTE#16#1B; (* ESC *)
    						x := x +1;
    						S_BUF.BUFFER[x] := BYTE#16#5B; (* [ *)
    						x := x +1;
    						S_BUF.BUFFER[x] := BYTE#16#30; (* 0 *)
    						x := x +1;
    						S_BUF.BUFFER[x] := BYTE#16#3B; (* ; *)
    						x := x +1;
    						S_BUF.BUFFER[x] := BYTE#16#33; (* 3 *)
    						x := x +1;
    						S_BUF.BUFFER[x] := (FRONT_COLOR AND BYTE#2#00000111) OR BYTE#16#30; (* Einerstelle Farbe Foreground ausgeben *)
    						x := x +1;
    						S_BUF.BUFFER[x] := BYTE#16#3B; (* ; *)
    						x := x +1;
    						S_BUF.BUFFER[x] := BYTE#16#34; (* 4 *)
    						x := x +1;
    						S_BUF.BUFFER[x] := (BACK_COLOR AND BYTE#2#00000111) OR BYTE#16#30; (* Einerstelle Farbe Background ausgeben *)
    						x := x +1;
    						S_BUF.BUFFER[x] := BYTE#16#6D; (* m *)
    					END_IF
    					(* Screen Clear *)
    					x := x +1;
    					S_BUF.BUFFER[x] := BYTE#16#1B; (* ESC *)
    					x := x +1;
    					S_BUF.BUFFER[x] := BYTE#16#5B; (* [ *)
    					x := x +1;
    					S_BUF.BUFFER[x] := BYTE#16#32; (* 2 *)
    					x := x +1;
    					S_BUF.BUFFER[x] := BYTE#16#4A; (* J *)
    				ELSE
    					x := x +1;
    					S_BUF.BUFFER[x] := BYTE#16#0A; (* neue Zeile *)
    				END_IF
    			END_IF

    			(* buffer voll , oder Daten sind vorhanden und kein weiterer Sendewunsch *)
    			IF (INT_TO_UINT(x + LEN(TEXT) + 21) > SIZEOF(S_BUF.BUFFER)) OR (x >= 0 AND NOT SEND) THEN
    				S_BUF.SIZE := INT_TO_UINT(x + 1); (* Länge eintragen -> Datensenden starten *)
    				x := -1;
    			ELSIF SEND THEN

    				(* aktuelle Farbe bestimmen  *)
    				IF b2_color AND FRONT_COLOR <> last_fc THEN
    					(* Farbeinstellung: ANSI-Sequenz ESC[x;Y;Zm ausgeben *)
    					x := x + 1;
    					S_BUF.BUFFER[x] := BYTE#16#1B; (* ESC *)
    					x := x + 1;
    					S_BUF.BUFFER[x] := BYTE#16#5B; (* [ *)
    					(* Farbeinstellung: dunkel oder Hell und blinken bestimmen *)
    					IF ((FRONT_COLOR AND BYTE#2#0001_1000) XOR (last_fc AND BYTE#2#0001_1000)) <> BYTE#00 OR TRUE THEN
    						x := x + 1;
    						S_BUF.BUFFER[x] := BYTE#16#30; (* 0  *)
    						x := x + 1;
    						S_BUF.BUFFER[x] := BYTE#16#3B; (* ; *)
    						(* keine dunklen Farben gewünscht -> dann Bold & Bright *)
    						IF (FRONT_COLOR AND BYTE#2#00001000) = BYTE#0 THEN
    							(* auf Bold & Bright Farben umstellen *)
    							x := x + 1;
    							S_BUF.BUFFER[x] := BYTE#16#31; (* 1 *)
    							x := x + 1;
    							S_BUF.BUFFER[x] := BYTE#16#3B; (* ; *)
    						END_IF
    						(* blinkenden Farben gewünscht *)
    						IF (FRONT_COLOR AND BYTE#2#00010000) > BYTE#0 THEN
    							(* auf Blinkenden Farbe umstellen *)
    							x := x + 1;
    							S_BUF.BUFFER[x] := BYTE#16#35; (* 5 *)
    							x := x + 1;
    							S_BUF.BUFFER[x] := BYTE#16#3B; (* ; *)
    						END_IF
    					END_IF
    					(* Zehnerstelle Farbe Foreground ausgeben *)
    					x := x + 1;
    					S_BUF.BUFFER[x] := BYTE#16#33; (* 3 *)
    					(* Einerstelle Farbe Foreground ausgeben *)
    					x := x + 1;
    					S_BUF.BUFFER[x] := (FRONT_COLOR AND BYTE#2#00000111) OR BYTE#16#30;
    					x := x + 1;
    					S_BUF.BUFFER[x] := BYTE#16#6D; (* m *)
    					(* neue Farbe als letzt verwendete speichern *)
    					last_fc := FRONT_COLOR;
    				END_IF

    				(* Cursor positionieren *)
    				IF X_POS > BYTE#0 AND Y_POS > BYTE#0 THEN
    					x := x + 1;
    					S_BUF.BUFFER[x] := BYTE#16#1B; (* ESC *)
    					x := x + 1;
    					S_BUF.BUFFER[x] := BYTE#16#5B; (* [ *)
    					(* Zehnerstelle Y_POS ausgeben *)
    					x := x + 1;
    					S_BUF.BUFFER[x] := SHR(INT_TO_BCDC(BYTE_TO_INT(Y_POS)),4) OR BYTE#16#30;
    					(* Einerstelle Y_POS ausgeben *)
    					x := x + 1;
    					S_BUF.BUFFER[x] := (INT_TO_BCDC(BYTE_TO_INT(Y_POS)) AND BYTE#16#0F) OR BYTE#16#30;
    					x := x + 1;
    					S_BUF.BUFFER[x] := BYTE#16#3B; (* ; *)
    					(* Zehnerstelle X_POS ausgeben *)
    					x := x + 1;
    					S_BUF.BUFFER[x] := SHR(INT_TO_BCDC(BYTE_TO_INT(X_POS)),4) OR BYTE#16#30;
    					(* Einerstelle X_POS ausgeben *)
    					x := x + 1;
    					S_BUF.BUFFER[x] := (INT_TO_BCDC(BYTE_TO_INT(X_POS)) AND BYTE#16#0F) OR BYTE#16#30;
    					x := x + 1;
    					S_BUF.BUFFER[x] := BYTE#16#48; (* H *)
    				END_IF

    				(* TEXT ausgeben *)
    				IF LEN(TEXT) > 0 THEN
    					_STRING_TO_BUFFER(str:=TEXT,pos:=x + 1,pt :=ADR(S_BUF.BUFFER), size:=SIZEOF(S_BUF.BUFFER));
    					x := x + LEN(TEXT);
    				END_IF

    				IF b3_cr_lr THEN (* OPTION: CR,LF ausgeben *)
    					x := x + 1;
    					S_BUF.BUFFER[x] := BYTE#16#0D;
    					x := x + 1;
    					S_BUF.BUFFER[x] := BYTE#16#0A;
    				END_IF

    				DONE := TRUE; (* Fertig in Buffer eingetragen *)

    				IF b7_no_flush THEN (* OPTION: no buffer flush *)
    					(* buffer sofort senden - aktuellen Schreibindex speichern -> Senden anstossen *)
    					S_BUF.SIZE := INT_TO_UINT(x + 1);
    					x := -1;
    				END_IF
    			END_IF
    		END_IF
    	END_IF
    END_CASE

    (* IP_FIFO *)
    IP_FIFO(FIFO:=IP_C.FIFO,state:=ip_state,ID:=ip_id);

    (* revision history
    ks	05. jan. 2009	rev 1.0
    	original version

    ks	20. oct. 2009	rev 1.1
    	Networkbuffer und Buffer-funktionen auf Basis 0

    ks	20. oct. 2009	rev 1.2
    	STRING(STRING_LENGTH)

    ks	17. may. 2011	rev 1.3
    	automatischer re-connect

    ks	03. dec. 2011	rev 1.4
    	initialisierung verbessert, PORT Nummer als Parmeter

    *)
END_FUNCTION_BLOCK

(* ---- TN_FRAMEWORK.st ---- *)
FUNCTION_BLOCK TN_FRAMEWORK
    (*http://www.oscat.de/images/OSCATNetwork/oscat_netlib121_en.pdf#page=173*)
    (* Initialisierung / Freigeben der Verbindung *)
    IF (NOT IP_C.C_ENABLE) THEN

    	(* IP Datenverkehr einrichten *)
    	IP_C.C_PORT := SEL(PORT=BYTE#0,PORT,WORD#23); (* Portnummer eintragen *)
    	IP_C.C_IP := DWORD#00; (* IP eintragen *)
    	IP_C.C_MODE := BYTE#4; (* Mode: TCP+PASSIV+PORT *)
    	IP_C.TIME_RESET := TRUE; (* Zeitueberwachung rücksetzen *)
    	IP_C.C_ENABLE := TRUE; (* Verbindungsaufbau freigeben *)
    	IP_C.R_OBSERVE := FALSE; (* keine Empfangsueberwachung *)

    END_IF

    t(IN:= IP_C.ERROR > DWORD#0, PT:=t#5s);
    IF t.Q THEN
    	IP_C.TIME_RESET := TRUE; (* Error Reset *)
    END_IF

    (* Telnet-Menu-Bar *)
    FB_TN_INPUT_MENU_BAR(
    	Xus_TN_MENU := US_TN_MENU,
    	Xus_TN_SCREEN := US_TN_SCREEN);

    (* Telnet-Input-Control *)
    FB_TN_INPUT_CONTROL(
    	Xus_TN_SCREEN := US_TN_SCREEN,
    	Xus_TN_INPUT_CONTROL := US_TN_INPUT_CONTROL);

    (* Telnet-Data-Send Line-Updates *)
    FB_TN_SEND_ROWS(
    	IP_C :=IP_C,
    	S_BUF :=S_BUF,
    	Xus_TN_SCREEN :=US_TN_SCREEN,
    	S_BUF_SIZE :=SIZEOF(S_BUF.BUFFER));

    (* Telnet-Server *)
    FB_IP_CONTROL(
    	IP_C :=IP_C,
    	S_BUF :=S_BUF,
    	R_BUF :=R_BUF,
    	IP :=DWORD#00,
    	PORT :=WORD#00,
    	TIME_OUT :=t#2s);

    (* Telnet-Data-Receive *)
    FB_TN_RECEIVE(
    	R_BUF := R_BUF,
    	Xus_TN_SCREEN := US_TN_SCREEN);

    (* revision history
    ks	10. mai. 2010	rev 1.0
    	original version

    ks	17. may. 2011	rev 1.1
    	automatischer re-connect

    ks	05. may. 2012	rev 1.2
    	neue parameter PORT
    *)
END_FUNCTION_BLOCK

(* ---- TN_INPUT_CONTROL.st ---- *)
FUNCTION_BLOCK TN_INPUT_CONTROL
    (*http://www.oscat.de/images/OSCATNetwork/oscat_netlib121_en.pdf#page=174*)
    (* Bearbeitung freigegeben ? *)
    IF (XUS_TN_INPUT_CONTROL.bo_Enable = FALSE) OR (XUS_TN_SCREEN.bo_Menue_Bar_Dialog = TRUE) THEN
    	RETURN;
    END_IF

    (* Fokus Reset durchführen *)
    IF (XUS_TN_INPUT_CONTROL.bo_Reset_Fokus = TRUE) THEN
    	XUS_TN_INPUT_CONTROL.bo_Reset_Fokus := FALSE;

    	FOR in_index := INT#01 TO XUS_TN_INPUT_CONTROL.in_Count DO
    		XUS_TN_INPUT_CONTROL.usa_TN_INPUT_CONTROL_DATA[in_index].bo_Focus := FALSE;
    	END_FOR

    	IF (XUS_TN_INPUT_CONTROL.in_Count >= INT#01) THEN
    		XUS_TN_INPUT_CONTROL.usa_TN_INPUT_CONTROL_DATA[1].bo_Focus := TRUE;
    		XUS_TN_INPUT_CONTROL.in_Focus_at := INT#01;
    	END_IF

    	XUS_TN_INPUT_CONTROL.bo_Update_all := TRUE;
    END_IF

    IF (XUS_TN_SCREEN.bo_Modal_Dialog = FALSE) THEN
    	(* TAB-Taste für Control-element wechsel auswerten *)
    	IF (XUS_TN_SCREEN.by_Input_Exten_Code = BYTE#09) THEN

    		in_Scroll_Offset := INT#01;

    		(* Cursor-Oben Taste *)
    	ELSIF (XUS_TN_SCREEN.by_Input_Exten_Code = BYTE#65) THEN

    		in_Scroll_Offset := -1;

    		(* Cursor-unten Taste *)
    	ELSIF (XUS_TN_SCREEN.by_Input_Exten_Code = BYTE#66) THEN

    		in_Scroll_Offset := INT#01;

    	END_IF
    END_IF

    IF (in_Scroll_Offset <> INT#00) THEN
    	(* Grenzwerte überprüfen                                            *)

    	XUS_TN_INPUT_CONTROL.in_Focus_at:=LIMIT(INT#01,XUS_TN_INPUT_CONTROL.in_Focus_at,XUS_TN_INPUT_CONTROL.in_Count);

    	in_Focus_new := XUS_TN_INPUT_CONTROL.in_Focus_at + in_Scroll_Offset;

    	IF (in_Focus_new > XUS_TN_INPUT_CONTROL.in_Count) THEN
    		in_Focus_new := INT#1;
    	END_IF

    	IF (in_Focus_new < INT#01) THEN
    		in_Focus_new := XUS_TN_INPUT_CONTROL.in_Count;
    	END_IF

    	in_Focus_alt := XUS_TN_INPUT_CONTROL.in_Focus_at;

    	(* aktuellen Element den Fokus entziehen *)
    	XUS_TN_INPUT_CONTROL.usa_TN_INPUT_CONTROL_DATA[in_Focus_alt].bo_Focus := FALSE;
    	XUS_TN_INPUT_CONTROL.usa_TN_INPUT_CONTROL_DATA[in_Focus_alt].bo_Update_Input := TRUE;

    	(* neuem Element den Fokus geben *)
    	XUS_TN_INPUT_CONTROL.usa_TN_INPUT_CONTROL_DATA[in_Focus_new].bo_Focus  := TRUE;
    	XUS_TN_INPUT_CONTROL.usa_TN_INPUT_CONTROL_DATA[in_Focus_new].bo_Update_Input := TRUE;

    	XUS_TN_INPUT_CONTROL.in_Focus_at := in_Focus_new;

    	bo_Tool_Tip_Update := TRUE;
    	in_Scroll_Offset := INT#00;

    END_IF

    (* Alle Elemente updaten ? *)
    IF (XUS_TN_INPUT_CONTROL.bo_Update_all = TRUE) THEN
    	FOR in_index := 1 TO XUS_TN_INPUT_CONTROL.in_Count DO
    		XUS_TN_INPUT_CONTROL.usa_TN_INPUT_CONTROL_DATA[in_index].bo_Update_All := TRUE;
    	END_FOR
    	XUS_TN_INPUT_CONTROL.bo_Update_all := FALSE;
    	bo_Tool_Tip_Update := TRUE;
    END_IF

    FOR in_index := 1 TO XUS_TN_INPUT_CONTROL.in_Count DO

    	IF (XUS_TN_INPUT_CONTROL.usa_TN_INPUT_CONTROL_DATA[in_index].in_Type > INT#00) THEN

    		IF (XUS_TN_INPUT_CONTROL.usa_TN_INPUT_CONTROL_DATA[in_index].bo_Focus = TRUE) THEN

    			XUS_TN_INPUT_CONTROL.usa_TN_INPUT_CONTROL_DATA[in_index].by_Input_ASCII_Code  := XUS_TN_SCREEN.by_Input_ASCII_Code;
    			XUS_TN_INPUT_CONTROL.usa_TN_INPUT_CONTROL_DATA[in_index].by_Input_Exten_Code  := XUS_TN_SCREEN.by_Input_Exten_Code;
    			XUS_TN_INPUT_CONTROL.usa_TN_INPUT_CONTROL_DATA[in_index].bo_Input_ASCII_IsNum := XUS_TN_SCREEN.bo_Input_ASCII_IsNum;

    			(* Tool-Tip Text ausgeben *)
    			IF (bo_Tool_Tip_Update = TRUE) THEN

    				FB_TN_SC_WRITE_C(	Iin_Y := XUS_TN_INPUT_CONTROL.in_ToolTip_Y,
    									Iin_X := XUS_TN_INPUT_CONTROL.in_ToolTip_X,
    									Iby_ATTR := XUS_TN_INPUT_CONTROL.by_ToolTip_Attr,
    									Iin_OPTION := INT#02, (* Center-String *)
    									Iin_LENGTH := XUS_TN_INPUT_CONTROL.in_ToolTip_Size,
    									Ist_STRING := XUS_TN_INPUT_CONTROL.usa_TN_INPUT_CONTROL_DATA[in_index].st_Input_ToolTip,
    									XUS_TN_SCREEN := XUS_TN_SCREEN);

    				(* Flag rücksetzen *)
    				bo_Tool_Tip_Update := FALSE;
    			END_IF
    		END_IF

    		CASE XUS_TN_INPUT_CONTROL.usa_TN_INPUT_CONTROL_DATA[in_index].in_Type OF
    		1:
    			(* Edit-Line bearbeiten *)
    			FB_TN_INPUT_EDIT_LINE(	Xus_TN_INPUT_CONTROL_DATA := XUS_TN_INPUT_CONTROL.usa_TN_INPUT_CONTROL_DATA[in_index],
    									XUS_TN_SCREEN := XUS_TN_SCREEN);
    		2:
    			(* Select-Text bearbeiten *)
    			FB_TN_INPUT_SELECT_TEXT(	Xus_TN_INPUT_CONTROL_DATA := XUS_TN_INPUT_CONTROL.usa_TN_INPUT_CONTROL_DATA[in_index],
    										XUS_TN_SCREEN := XUS_TN_SCREEN);
    		3:
    			(* Select-Popup bearbeiten *)
    			FB_TN_INPUT_SELECT_POPUP(	Xus_TN_INPUT_CONTROL_DATA := XUS_TN_INPUT_CONTROL.usa_TN_INPUT_CONTROL_DATA[in_index],
    										XUS_TN_SCREEN := XUS_TN_SCREEN);
    		END_CASE

    		IF (XUS_TN_INPUT_CONTROL.usa_TN_INPUT_CONTROL_DATA[in_index].bo_Focus = TRUE) THEN

    			(* Cursor position von Element auf Screen übertragen *)
    			XUS_TN_SCREEN.in_Cursor_X := XUS_TN_INPUT_CONTROL.usa_TN_INPUT_CONTROL_DATA[in_index].in_Cursor_X;
    			XUS_TN_SCREEN.in_Cursor_Y := XUS_TN_INPUT_CONTROL.usa_TN_INPUT_CONTROL_DATA[in_index].in_Cursor_Y;

    		END_IF
    	END_IF
    END_FOR

    (* revision history
    ks	10. mai. 2010	rev 1.0
    	original version
    *)
END_FUNCTION_BLOCK

(* ---- TN_INPUT_EDIT_LINE.st ---- *)
FUNCTION_BLOCK TN_INPUT_EDIT_LINE
    (*http://www.oscat.de/images/OSCATNetwork/oscat_netlib121_en.pdf#page=174*)
    (* Cursorsteuerung rücksetzen *)
    in_CursorOffset := INT#0;

    IF XUS_TN_INPUT_CONTROL_DATA.bo_Focus = TRUE THEN

    	(* Texteingabe erkannt ? *)
    	IF XUS_TN_INPUT_CONTROL_DATA.by_Input_ASCII_Code > BYTE#0 THEN

    		IF (XUS_TN_INPUT_CONTROL_DATA.bo_Input_Only_Num = TRUE AND XUS_TN_INPUT_CONTROL_DATA.bo_Input_ASCII_IsNum = TRUE)
    			OR (XUS_TN_INPUT_CONTROL_DATA.bo_Input_Only_Num = FALSE) THEN

    			(* ASCII Wert in einen String wandeln *)
    			st_CHAR := CHR_TO_STRING(C:=XUS_TN_INPUT_CONTROL_DATA.by_Input_ASCII_Code);

    			(* Eingabe übernehmen *)
    			XUS_TN_INPUT_CONTROL_DATA.st_Input_Data := REPLACE(XUS_TN_INPUT_CONTROL_DATA.st_Input_Data,
    			st_CHAR,INT#1,XUS_TN_INPUT_CONTROL_DATA.in_Cursor_Pos);

    			in_CursorOffset := INT#1;
    			XUS_TN_INPUT_CONTROL_DATA.bo_Update_Input := TRUE;
    		END_IF
    	END_IF

    	CASE BYTE_TO_INT(XUS_TN_INPUT_CONTROL_DATA.by_Input_Exten_Code) OF

    	67: (* Cursor rechts gedrückt *)
    		in_CursorOffset := INT#1;

    	68: (* Cursor links gedrückt *)
    		in_CursorOffset := -1;

    	08: (* Backspace gedrückt *)
    		XUS_TN_INPUT_CONTROL_DATA.st_Input_Data := REPLACE(XUS_TN_INPUT_CONTROL_DATA.st_Input_Data, ' ', 1,XUS_TN_INPUT_CONTROL_DATA.in_Cursor_Pos);
    		XUS_TN_INPUT_CONTROL_DATA.bo_Update_Input := TRUE;
    		in_CursorOffset := -1;

    	13: (* Enter-Taste gedrückt *)
    		IF LEN(XUS_TN_INPUT_CONTROL_DATA.st_Input_Mask) > INT#00 THEN
    			(* Eingabestring übernehmen *)
    			XUS_TN_INPUT_CONTROL_DATA.st_Input_String := XUS_TN_INPUT_CONTROL_DATA.st_Input_Data;

    			(* Eingabestring -> links und rechts Leerzeichen entfernen *)
    			XUS_TN_INPUT_CONTROL_DATA.st_Input_String := TRIME(str:=XUS_TN_INPUT_CONTROL_DATA.st_Input_String);
    			XUS_TN_INPUT_CONTROL_DATA.bo_Input_Entered := TRUE;

    			(* neue Eingabe vorbereiten *)
    			XUS_TN_INPUT_CONTROL_DATA.st_Input_Data := XUS_TN_INPUT_CONTROL_DATA.st_Input_Mask;

    			XUS_TN_INPUT_CONTROL_DATA.in_Cursor_Pos := INT#1;
    			XUS_TN_INPUT_CONTROL_DATA.bo_Update_Input := TRUE;

    			(* suche erstes Position in Eingabemaske *)
    			st_CHAR := MID(XUS_TN_INPUT_CONTROL_DATA.st_Input_Mask,1,XUS_TN_INPUT_CONTROL_DATA.in_Cursor_Pos);
    			IF st_CHAR <> ' ' THEN
    				(* nächsten Eingabeposition suchen *)
    				in_CursorOffset := INT#1;
    			END_IF
    		END_IF
    	END_CASE
    END_IF

    (* Cursor richtung rechts bewegen                                   *)
    IF (in_CursorOffset > INT#0) OR (XUS_TN_INPUT_CONTROL_DATA.in_Cursor_Pos = INT#0) THEN
    	bo_Pos_Found := FALSE;

    	in_count := XUS_TN_INPUT_CONTROL_DATA.in_Cursor_Pos + INT#1;
    	in_Count_End := LEN(XUS_TN_INPUT_CONTROL_DATA.st_Input_Mask);

    	WHILE (in_count <= in_Count_End) AND (bo_Pos_Found = FALSE) DO

    		st_CHAR := MID(XUS_TN_INPUT_CONTROL_DATA.st_Input_Mask,1,in_count);
    		IF st_CHAR = ' ' THEN
    			XUS_TN_INPUT_CONTROL_DATA.in_Cursor_Pos := in_count;
    			XUS_TN_INPUT_CONTROL_DATA.bo_Update_Input := TRUE;
    			bo_Pos_Found := TRUE;
    		END_IF

    		in_count := in_count + INT#1;

    	END_WHILE
    END_IF

    (* Cursor richtung links bewegen *)
    IF in_CursorOffset < INT#0 THEN
    	bo_Pos_Found := FALSE;

    	in_count     := XUS_TN_INPUT_CONTROL_DATA.in_Cursor_Pos - INT#01;
    	in_Count_End := INT#1;

    	WHILE (in_count >= in_Count_End) AND (bo_Pos_Found = FALSE) DO

    		st_CHAR := MID(XUS_TN_INPUT_CONTROL_DATA.st_Input_Mask,1,in_count);
    		IF st_CHAR = ' ' THEN
    			XUS_TN_INPUT_CONTROL_DATA.in_Cursor_Pos := in_count;
    			XUS_TN_INPUT_CONTROL_DATA.bo_Update_Input := TRUE;
    			bo_Pos_Found := TRUE;
    		END_IF

    		in_count := in_count - INT#1;
    	END_WHILE
    END_IF

    (* maximale Cursorposition ? *)
    IF XUS_TN_INPUT_CONTROL_DATA.in_Cursor_Pos > LEN(XUS_TN_INPUT_CONTROL_DATA.st_Input_Data) THEN
    	XUS_TN_INPUT_CONTROL_DATA.in_Cursor_Pos := LEN(XUS_TN_INPUT_CONTROL_DATA.st_Input_Data);
    	XUS_TN_INPUT_CONTROL_DATA.bo_Update_Input := TRUE;
    END_IF

    (* minimale Cursorposition ? *)
    IF XUS_TN_INPUT_CONTROL_DATA.in_Cursor_Pos < INT#1 THEN
    	XUS_TN_INPUT_CONTROL_DATA.in_Cursor_Pos := INT#1;
    	XUS_TN_INPUT_CONTROL_DATA.bo_Update_Input := TRUE;
    END_IF

    (* Aktualisierung der Anzeige *)
    IF (XUS_TN_INPUT_CONTROL_DATA.bo_Update_Input = TRUE) OR (XUS_TN_INPUT_CONTROL_DATA.bo_Update_All = TRUE) THEN

    	(* Title-Text ausgeben *)
    	IF (XUS_TN_INPUT_CONTROL_DATA.bo_Update_All = TRUE) THEN

    		IF (XUS_TN_INPUT_CONTROL_DATA.in_Title_X_Offset = INT#00) AND (XUS_TN_INPUT_CONTROL_DATA.in_Title_Y_Offset = INT#00) THEN
    			(* wenn Offset X,Y =0 dann Titlestring links vom Element positionieren *)
    			FB_TN_SC_WRITE.Iin_Y := XUS_TN_INPUT_CONTROL_DATA.in_Y;
    			FB_TN_SC_WRITE.Iin_X := XUS_TN_INPUT_CONTROL_DATA.in_X - LEN(XUS_TN_INPUT_CONTROL_DATA.st_Title_String);
    		ELSE
    			(* Title-Text durch Row, Color-Offset ausgeben *)
    			FB_TN_SC_WRITE.Iin_Y := XUS_TN_INPUT_CONTROL_DATA.in_Y + XUS_TN_INPUT_CONTROL_DATA.in_Title_Y_Offset;
    			FB_TN_SC_WRITE.Iin_X := XUS_TN_INPUT_CONTROL_DATA.in_X + XUS_TN_INPUT_CONTROL_DATA.in_Title_X_Offset;
    		END_IF

    		(* Title-Text durch Row, Color-Offset ausgeben *)
    		FB_TN_SC_WRITE(	Iby_ATTR := XUS_TN_INPUT_CONTROL_DATA.by_Title_Attr,
    						Ist_STRING := XUS_TN_INPUT_CONTROL_DATA.st_Title_String,
    						XUS_TN_SCREEN := XUS_TN_SCREEN);
    	END_IF

    	(* Eingabetext ausgeben *)
    	IF (XUS_TN_INPUT_CONTROL_DATA.bo_Input_Hidden = TRUE) THEN

    		st_String := '';

    		IF LEN(XUS_TN_INPUT_CONTROL_DATA.st_Input_Data) = LEN(XUS_TN_INPUT_CONTROL_DATA.st_Input_Mask) THEN
    			(* Eingabemodus: HIDDEN *)
    			FOR in_count := 1 TO LEN(XUS_TN_INPUT_CONTROL_DATA.st_Input_Data) DO

    				(* Zeichen aus Eingabemaske lesen *)
    				st_CHAR := MID(XUS_TN_INPUT_CONTROL_DATA.st_Input_Mask,1,in_count);

    				(* Eingabe oder Maskenzeichen ausgeben *)
    				IF st_CHAR = ' ' THEN

    					(* Zeichen aus Eingabedata lesen *)
    					st_CHAR := MID(XUS_TN_INPUT_CONTROL_DATA.st_Input_Data,1,in_count);

    					IF st_CHAR = ' ' THEN
    						(* Leerzeichen ausgeben *)
    						st_String := CONCAT(st_String, ' ');

    					ELSE
    						(* verdecktes Zeichen ausgeben *)
    						st_String := CONCAT(st_String, '*');

    					END_IF

    				ELSE
    					(* Zeichen aus Eingabemaske übernehmen *)
    					st_CHAR := MID(XUS_TN_INPUT_CONTROL_DATA.st_Input_Data,1,in_count);
    					st_String := CONCAT(st_String,st_CHAR);

    				END_IF
    			END_FOR
    		END_IF
    	ELSE

    		(* Eingabemodus: NORMAL *)
    		st_String := XUS_TN_INPUT_CONTROL_DATA.st_Input_Data;

    	END_IF

    	(* String ausgeben *)

    	IF XUS_TN_INPUT_CONTROL_DATA.bo_Focus = TRUE THEN
    		by_Attr := XUS_TN_INPUT_CONTROL_DATA.by_Attr_mF;
    	ELSE
    		by_Attr := XUS_TN_INPUT_CONTROL_DATA.by_Attr_oF;
    	END_IF

    	FB_TN_SC_WRITE(	Iin_Y := XUS_TN_INPUT_CONTROL_DATA.in_Y,
    					Iin_X := XUS_TN_INPUT_CONTROL_DATA.in_X,
    					Iby_ATTR := by_Attr,
    					Ist_STRING := st_String,
    					XUS_TN_SCREEN := XUS_TN_SCREEN);

    	(* Cursor auf aktuelle Position setzen *)
    	XUS_TN_INPUT_CONTROL_DATA.in_Cursor_Y := XUS_TN_INPUT_CONTROL_DATA.in_Y;
    	XUS_TN_INPUT_CONTROL_DATA.in_Cursor_X := XUS_TN_INPUT_CONTROL_DATA.in_X + XUS_TN_INPUT_CONTROL_DATA.in_Cursor_Pos - INT#1;

    	in_old_charpos := INT#0;

    	(* Update-Flag's rücksetzen *)
    	XUS_TN_INPUT_CONTROL_DATA.bo_Update_All := FALSE;
    	XUS_TN_INPUT_CONTROL_DATA.bo_Update_Input := FALSE;
    END_IF

    (* revision history
    ks	10. mai. 2010	rev 1.0
    	original version
    *)
END_FUNCTION_BLOCK

(* ---- TN_INPUT_MENU_BAR.st ---- *)
FUNCTION_BLOCK TN_INPUT_MENU_BAR
    (*http://www.oscat.de/images/OSCATNetwork/oscat_netlib121_en.pdf#page=176*)
    (* sicherstellen das rechteck immer innerhalb screen positioniert wird *)

    IF (XUS_TN_MENU.in_State = INT#00) AND (XUS_TN_MENU.bo_Create = TRUE) THEN
    	XUS_TN_MENU.in_State := INT#01;
    	XUS_TN_MENU.bo_Create := FALSE;
    	XUS_TN_MENU.in_Menu_Selected := INT#00;
    	XUS_TN_MENU.bo_Update := TRUE;
    	bo_Reset_Position := TRUE;

    	(* Menu-Bar - Hauptmenue *)
    	st_MENU_BAR := ELEMENT_GET(SEP:=BYTE#37,POS:=0,ELEMENT:=XUS_TN_MENU.st_MENU_TEXT);

    	(* Menu-Bar - Anzahl der Elemente bestimmen *)
    	XUS_TN_MENU.in_Menu_E_Count := ELEMENT_COUNT(SEP:=BYTE#35,ELEMENT:=st_MENU_BAR);

    END_IF

    (* Keycode ablegen *)
    by_New_KeyCode := XUS_TN_SCREEN.by_Input_Exten_Code;

    (* Popup-Menu Tastensteuerung (nur Cursor oben + unten zulassen *)
    IF (by_New_KeyCode = BYTE#65) OR (by_New_KeyCode = BYTE#66) THEN
    	us_TN_MENU_POPUP.by_Input_Exten_Code := by_New_KeyCode;
    ELSE
    	us_TN_MENU_POPUP.by_Input_Exten_Code := BYTE#00;
    END_IF

    (* Escape *)
    IF (by_New_KeyCode = BYTE#27) THEN
    	(* Menu war inaktiv -> Escape -> Menu aktivieren *)
    	IF (XUS_TN_MENU.in_State = INT#01) AND (XUS_TN_SCREEN.bo_Modal_Dialog = FALSE) THEN
    		XUS_TN_MENU.in_State := INT#02;
    		XUS_TN_MENU.bo_Update := TRUE;
    		XUS_TN_MENU.in_Menu_Selected := INT#00;

    		XUS_TN_SCREEN.bo_Menue_Bar_Dialog := TRUE;

    		(* Menu war aktiv -> Escape -> Menu deaktivieren *)
    	ELSIF (XUS_TN_MENU.in_State = INT#02) THEN
    		us_TN_MENU_POPUP.bo_Destroy := TRUE;
    		XUS_TN_MENU.bo_Update := TRUE;
    		XUS_TN_MENU.in_State := INT#01;
    		bo_Reset_Position := TRUE;

    		XUS_TN_SCREEN.bo_Menue_Bar_Dialog := FALSE;
    	END_IF
    END_IF

    (* Menu aktiv *)
    IF (XUS_TN_MENU.in_State = INT#02) THEN

    	(* Return *)
    	IF (by_New_KeyCode = BYTE#13)  THEN
    		us_TN_MENU_POPUP.bo_Destroy := TRUE;
    		XUS_TN_MENU.bo_Update := TRUE;
    		XUS_TN_MENU.in_State := INT#01;
    		bo_Reset_Position := TRUE;
    		XUS_TN_MENU.in_Menu_Selected := (XUS_TN_MENU.in_Cur_Menu_Item * INT#10) + XUS_TN_MENU.in_Cur_Sub_Item;
    		XUS_TN_SCREEN.by_Input_Exten_Code := BYTE#00;

    		XUS_TN_SCREEN.bo_Menue_Bar_Dialog := FALSE;

    		(* Destroy-Befehl -> Popup-Menu beenden *)
    	ELSIF (XUS_TN_MENU.bo_Destroy = TRUE) THEN
    		us_TN_MENU_POPUP.bo_Destroy := TRUE;
    		XUS_TN_MENU.bo_Update := TRUE;
    		XUS_TN_MENU.in_State := INT#01;
    		bo_Reset_Position := TRUE;
    		XUS_TN_MENU.in_Menu_Selected := INT#00;
    		XUS_TN_SCREEN.by_Input_Exten_Code := BYTE#00;

    		XUS_TN_SCREEN.bo_Menue_Bar_Dialog := FALSE;

    	END_IF

    	IF (by_New_KeyCode = BYTE#67) THEN (* Cursor rechts *)
    		in_Scroll_Offset := INT#1;
    		XUS_TN_MENU.bo_Update := TRUE;
    		XUS_TN_SCREEN.by_Input_Exten_Code := BYTE#00;

    	ELSIF (by_New_KeyCode = BYTE#68) THEN (* Cursor links *)
    		in_Scroll_Offset := -1;
    		XUS_TN_MENU.bo_Update := TRUE;
    		XUS_TN_SCREEN.by_Input_Exten_Code := BYTE#00;
    	END_IF
    END_IF

    IF bo_Reset_Position = TRUE THEN
    	bo_Reset_Position := FALSE;
    	XUS_TN_MENU.in_X_SM_old := -1;
    	XUS_TN_MENU.in_Y_SM_old := -1;
    	XUS_TN_MENU.in_X_SM_new := -1;
    	XUS_TN_MENU.in_Y_SM_new := -1;
    END_IF

    (* POPUP-Menu updaten *)
    IF (XUS_TN_MENU.in_State > INT#00) AND (XUS_TN_MENU.bo_Update = TRUE) THEN

    	XUS_TN_MENU.bo_Update := FALSE;

    	in_ROW := XUS_TN_MENU.in_Y;
    	in_COL := XUS_TN_MENU.in_X;

    	(* Scrolloffset *)
    	IF in_Scroll_Offset <> INT#00 THEN
    		XUS_TN_MENU.in_Cur_Menu_Item := INC2(XUS_TN_MENU.in_Cur_Menu_Item,in_Scroll_Offset,1,XUS_TN_MENU.in_Menu_E_Count);
    		in_Scroll_Offset := INT#00;
    	ELSE
    		(* Item = 0 und kein Scrolloffset *)
    		IF (XUS_TN_MENU.in_Cur_Menu_Item = INT#00) THEN
    			XUS_TN_MENU.in_Cur_Menu_Item := INT#01;
    		END_IF
    	END_IF

    	(* alle Menutext zeichnen *)
    	FOR in_Count := INT#01 TO XUS_TN_MENU.in_Menu_E_Count DO;

    		(* Zeichenfarbe bestimmen *)
    		IF (in_Count = XUS_TN_MENU.in_Cur_Menu_Item) AND (XUS_TN_MENU.in_State > INT#01 ) THEN
    			by_ATTR := XUS_TN_MENU.by_Attr_mF;

    			XUS_TN_MENU.in_Y_SM_new := in_ROW + INT#01;
    			XUS_TN_MENU.in_X_SM_new := in_COL;

    		ELSE
    			by_ATTR := XUS_TN_MENU.by_Attr_oF;
    		END_IF

    		st_MENU_TITLE := ELEMENT_GET(SEP:=BYTE#35,POS:=in_Count - 1,ELEMENT:=st_MENU_BAR);

    		in_TITLE_Length := LEN(st_MENU_TITLE) + INT#02;

    		FB_TN_SC_WRITE_C(	Iin_Y := in_ROW,
    							Iin_X := in_COL,
    							Iby_ATTR := by_ATTR,
    							Iin_LENGTH := in_TITLE_Length,
    							Iin_OPTION := INT#02,
    							Ist_STRING := st_MENU_TITLE,
    							XUS_TN_SCREEN := XUS_TN_SCREEN);

    		in_COL := in_COL + in_TITLE_Length;

    	END_FOR
    END_IF

    IF XUS_TN_MENU.in_X_SM_new <> XUS_TN_MENU.in_X_SM_old THEN

    	(* SubMenu ist aktiv -> beenden                                     *)
    	IF us_TN_MENU_POPUP.bo_Activ = TRUE THEN
    		us_TN_MENU_POPUP.bo_Destroy := TRUE;

    		(* Sub-Menu bearbeiten *)
    		FB_TN_INPUT_MENU_POPUP(	Xus_TN_MENU_POPUP := us_TN_MENU_POPUP,
    								XUS_TN_SCREEN := XUS_TN_SCREEN);
    	END_IF

    	IF us_TN_MENU_POPUP.bo_Activ = FALSE THEN
    		(* Popup-Menu zu aktuellen Menu parametrieren und ausführen         *)
    		in_Index := XUS_TN_MENU.in_Cur_Menu_Item;

    		us_TN_MENU_POPUP.in_Y := XUS_TN_MENU.in_Y_SM_new;
    		us_TN_MENU_POPUP.in_X := XUS_TN_MENU.in_X_SM_new;
    		us_TN_MENU_POPUP.by_Attr_mF := XUS_TN_MENU.by_Attr_mF;
    		us_TN_MENU_POPUP.by_Attr_oF := XUS_TN_MENU.by_Attr_oF;
    		us_TN_MENU_POPUP.st_Menu_Text := ELEMENT_GET(SEP:=BYTE#37,POS:=in_Index,ELEMENT:=XUS_TN_MENU.st_MENU_TEXT);
    		us_TN_MENU_POPUP.bo_Create := TRUE;

    		XUS_TN_MENU.in_X_SM_old := XUS_TN_MENU.in_X_SM_new;
    		XUS_TN_MENU.in_Y_SM_old := XUS_TN_MENU.in_Y_SM_new;

    	END_IF
    END_IF

    (* Popup-Menu zyklisch aufrufen *)
    FB_TN_INPUT_MENU_POPUP(	Xus_TN_MENU_POPUP := us_TN_MENU_POPUP,
    						XUS_TN_SCREEN := XUS_TN_SCREEN);

    (* aktuelles Item vom Popup-Menu kopieren *)
    XUS_TN_MENU.in_Cur_Sub_Item := us_TN_MENU_POPUP.in_Cur_Item;

    (* Destroy-Befehl *)
    IF (XUS_TN_MENU.in_State = INT#01) THEN
    	IF (XUS_TN_MENU.bo_Destroy = TRUE) THEN
    		XUS_TN_MENU.in_State := INT#00;
    		XUS_TN_MENU.bo_Destroy := FALSE;
    		XUS_TN_MENU.in_Cur_Menu_Item := INT#00;
    		XUS_TN_MENU.in_Cur_Sub_Item := INT#00;
    	END_IF
    END_IF

    (* revision history
    ks	06. apr. 2011	rev 1.1
    	list_len und list_get durch element_count und element_get ersetzt

    ks	10. mai. 2010	rev 1.0
    	original version
    *)
END_FUNCTION_BLOCK
